	HUS2_VP1_MQ41_ID	AT%MB2524	:REAL;	(*	HUS2_VP1_MQ41_ID	AS01	GVL.HUS2_VP1_MQ41_ID	REAL							Mätar-ID VP1-MQ41			*)
	HUS2_VP1_MQ41_GT41_MV	AT%MB2528	:REAL;	(*	HUS2_VP1_MQ41_GT41_MV	AS01	GVL.HUS2_VP1_MQ41_GT41_MV	REAL	-50	150	-50	150	°C	0.0	Framledningstemperatur fjärrvärme			*)					
	HUS2_VP1_MQ41_GT42_MV	AT%MB2532	:REAL;	(*	HUS2_VP1_MQ41_GT42_MV	AS01	GVL.HUS2_VP1_MQ41_GT42_MV	REAL	-50	150	-50	150	°C	0.0	Returtemperatur fjärrvärme			*)					
	HUS2_VP1_MQ41_DLT	AT%MB2536	:REAL;	(*	HUS2_VP1_MQ41_DLT	AS01	GVL.HUS2_VP1_MQ41_DLT	REAL	-50	150	-50	150	°C	0.0	Temperaturdifferens fjärrvärme			*)					
	HUS2_VP1_MQ41_P	AT%MB2540	:REAL;	(*	HUS2_VP1_MQ41_P	AS01	GVL.HUS2_VP1_MQ41_P	REAL	0	1000	0	1000	Kw	0.0	Momentant effektuttag			*)					
	HUS2_VP1_MQ41_Q	AT%MB2544	:REAL;	(*	HUS2_VP1_MQ41_Q	AS01	GVL.HUS2_VP1_MQ41_Q	REAL	0				m3/h	0.0	Momentant flöde			*)					
	HUS2_VP1_MQ41_E	AT%MB2548	:REAL;	(*	HUS2_VP1_MQ41_E	AS01	GVL.HUS2_VP1_MQ41_E	REAL	0				MWh	0.0	Total energiförbrukning			*)					
																							
	HUS2_VS1_GT11_BB	AT%MB2552	:REAL;	(*	HUS2_VS1_GT11_BB	AS01	GVL.HUS2_VS1_GT11_BB	REAL	0	150	0	150	°C	0.0	Beräknat börvärde framledningstemperatur			*)
	HUS2_VP1_MQ41_BB	AT%MB2556	:REAL;	(*	HUS2_VP1_MQ41_BB	AS01	GVL.HUS2_VP1_MQ41_BB	REAL	0	500	0	500	kWh	0.0	Beräknad maxeffekt			*)				

																							
																							

																						
																						


																					

END_VAR

(* Global variable list: HUS2/VS30/HUS2_VS30_INST *)
VAR_GLOBAL PERSISTENT


					(*	Name	Device	Address	Data type	Rawmin	Rawmax	Engmin	Engmax	Unit	Format	Description	Alarmoptions	Trendoptions	*)
																								
		HUS2_VS30_GT11_UX1	AT%MB2700	:REAL;	(*	HUS2_VS30_GT11_UX1	AS01	GVL.HUS2_VS30_GT11_UX1	REAL	-50	150	-50	150	°C	0.0	Utetemp. kompenserad kurva Brytpunkt X1			*)					
		HUS2_VS30_GT11_UX2	AT%MB2704	:REAL;	(*	HUS2_VS30_GT11_UX2	AS01	GVL.HUS2_VS30_GT11_UX2	REAL	-50	150	-50	150	°C	0.0	Utetemp. kompenserad kurva Brytpunkt X2			*)					
		HUS2_VS30_GT11_UX3	AT%MB2708	:REAL;	(*	HUS2_VS30_GT11_UX3	AS01	GVL.HUS2_VS30_GT11_UX3	REAL	-50	150	-50	150	°C	0.0	Utetemp. kompenserad kurva Brytpunkt X3			*)					
		HUS2_VS30_GT11_UX4	AT%MB2712	:REAL;	(*	HUS2_VS30_GT11_UX4	AS01	GVL.HUS2_VS30_GT11_UX4	REAL	-50	150	-50	150	°C	0.0	Utetemp. kompenserad kurva Brytpunkt X4			*)					
		HUS2_VS30_GT11_UX5	AT%MB2716	:REAL;	(*	HUS2_VS30_GT11_UX5	AS01	GVL.HUS2_VS30_GT11_UX5	REAL	-50	150	-50	150	°C	0.0	Utetemp. kompenserad kurva Brytpunkt X5			*)					
		HUS2_VS30_GT11_UY1	AT%MB2720	:REAL;	(*	HUS2_VS30_GT11_UY1	AS01	GVL.HUS2_VS30_GT11_UY1	REAL	0	150	0	150	°C	0.0	Utetemp. kompenserad kurva Brytpunkt Y1			*)					
		HUS2_VS30_GT11_UY2	AT%MB2724	:REAL;	(*	HUS2_VS30_GT11_UY2	AS01	GVL.HUS2_VS30_GT11_UY2	REAL	0	150	0	150	°C	0.0	Utetemp. kompenserad kurva Brytpunkt Y2			*)					
		HUS2_VS30_GT11_UY3	AT%MB2728	:REAL;	(*	HUS2_VS30_GT11_UY3	AS01	GVL.HUS2_VS30_GT11_UY3	REAL	0	150	0	150	°C	0.0	Utetemp. kompenserad kurva Brytpunkt Y3			*)					
		HUS2_VS30_GT11_UY4	AT%MB2732	:REAL;	(*	HUS2_VS30_GT11_UY4	AS01	GVL.HUS2_VS30_GT11_UY4	REAL	0	150	0	150	°C	0.0	Utetemp. kompenserad kurva Brytpunkt Y4			*)					
		HUS2_VS30_GT11_UY5	AT%MB2736	:REAL;	(*	HUS2_VS30_GT11_UY5	AS01	GVL.HUS2_VS30_GT11_UY5	REAL	0	150	0	150	°C	0.0	Utetemp. kompenserad kurva Brytpunkt Y5			*)					
		HUS2_VS30_GT11_UMIN	AT%MB2740	:REAL;	(*	HUS2_VS30_GT11_UMIN	AS01	GVL.HUS2_VS30_GT11_UMIN	REAL	0	150	0	150	°C	0.0	Utetemp. kompenserad kurva Min-begränsning			*)					
		HUS2_VS30_GT11_UMAX	AT%MB2744	:REAL;	(*	HUS2_VS30_GT11_UMAX	AS01	GVL.HUS2_VS30_GT11_UMAX	REAL	0	150	0	150	°C	0.0	Utetemp. kompenserad kurva Max-begränsning			*)					
																								
		HUS2_VS30_GT11_CP	AT%MB2748	:REAL;	(*	HUS2_VS30_GT11_CPV	AS01	GVL.HUS2_VS30_GT11_CP	REAL	0	10	0	10		0.0	P-parameter			*)					
		HUS2_VS30_GT11_CI	AT%MB2752	:REAL;	(*	HUS2_VS30_GT11_CIV	AS01	GVL.HUS2_VS30_GT11_CI	REAL	0	900	0	900	Sek		I-Tid 			*)
		HUS2_VS30_GT11_CD	AT%MB2756	:REAL;	(*	HUS2_VS30_GT11_CDV	AS01	GVL.HUS2_VS30_GT11_CD	REAL	0	900	0	900	Sek		D-tid 			*)
		HUS2_VS30_GT11_CS	AT%MB2760	:REAL;	(*	HUS2_VS30_GT11_CSV	AS01	GVL.HUS2_VS30_GT11_CS	REAL	0	900	0	900	Sek		Samplingstid			*)
		HUS2_VS30_GT11_CZ	AT%MB2764	:REAL;	(*	HUS2_VS30_GT11_CZV	AS01	GVL.HUS2_VS30_GT11_CZ	REAL	-10	10	-10	10	°C	0.0	Dödband regulator			*)					
																								
		HUS2_VS30_SO1_MAN	AT%MB2768	:INT;	(*	HUS2_VS30_SO1_MAN	AS01	GVL.HUS2_VS30_SO1_MAN	INT	0	2	0	2			Manuell styrning system VS30. 0=Auto, 1=Manuell från, 2=Manuell till			*)					
		HUS2_VS30_PV01_MAN	AT%MB2770	:INT;	(*	HUS2_VS30_PV01_MAN	AS01	GVL.HUS2_VS30_PV01_MAN	INT	0	2	0	2			Manuell styrning crikulationspump 0=Auto,1=Från,2=Till			*)					
		HUS2_VS30_SV21_MAN1	AT%MB2772	:INT;	(*	HUS2_VS30_SV21_MAN	AS01	GVL.HUS2_VS30_SV21_MAN	INT	0	1	0	1			Manuell styrning ventilställdon 0=Auto,1=Hand			*)					
		HUS2_VS30_SV21_RMAN	AT%MB2776	:REAL;	(*	HUS2_VS30_SV21_RMAN	AS01	GVL.HUS2_VS30_SV21_RMAN	REAL	0	100	0	100	%		Manuell styrsignal ventilställdon			*)					
																								
		HUS2_VS30_SO1_FLM	AT%MB2780	:INT;	(*	HUS2_VS30_SO1_FLM	AS01	GVL.HUS2_VS30_SO1_FLM	INT	0	3600	0	3600	Min		Larmfördröjning serviceomkopplare ej i läge AUTO			*)					
		HUS2_VS30_PV01_FLM	AT%MB2782	:INT;	(*	HUS2_VS30_PV01_FLM	AS01	GVL.HUS2_VS30_PV01_FLM	INT	0	3600	0	3600	Min		Larmfördröjning cirkulationspump ej i AUTO			*)					
		HUS2_VS30_SV21_FLM	AT%MB2784	:INT;	(*	HUS2_VS30_SV21_FLM	AS01	GVL.HUS2_VS30_SV21_FLM	INT	0	3600	0	3600	Min		Larmfördröjning ventilställdon ej i AUTO			*)					
		HUS2_VS30_PV01_FLD	AT%MB2786	:INT;	(*	HUS2_VS30_PV01_FLD	AS01	GVL.HUS2_VS30_PV01_FLD	INT	0	120	0	120	Sek		Larmfördröjning driftfel cirkulationspump			*)					
																								
		HUS2_VS30_GT11_GAVH	AT%MB2788	:REAL;	(*	HUS2_VS30_GT11_GAVH	AS01	GVL.HUS2_VS30_GT11_GAVH	REAL	-20	20	-20	20	°C	0.0	Gränsavvikelse hög framledningstemperatur			*)					
		HUS2_VS30_GT11_GAVL	AT%MB2792	:REAL;	(*	HUS2_VS30_GT11_GAVL	AS01	GVL.HUS2_VS30_GT11_GAVL	REAL	-20	20	-20	20	°C	0.0	Gränsavvikelse låg framledningstemperatur			*)					
		HUS2_VS30_GT11_FLAH	AT%MB2796	:INT;	(*	HUS2_VS30_GT11_FLAH	AS01	GVL.HUS2_VS30_GT11_FLAH	INT	0	3600	0	3600	Min		Larmfördröjning hög framledningstemperatur			*)					
		HUS2_VS30_GT11_FLAL	AT%MB2798	:INT;	(*	HUS2_VS30_GT11_FLAL	AS01	GVL.HUS2_VS30_GT11_FLAL	INT	0	3600	0	3600	Min		Lamfördröjning låg framledningstemperatur			*)					


																								

																								
		HUS2_VS30_GT11_KRV	AT%MB2816	:REAL;	(*	HUS2_VS30_GT11_KRV	AS01	GVL.HUS2_VS30_GT11_KRV	REAL	-10	10	-10	10	°C	0.0	Kalibreringsvärde framledningsgivare			*)					
		HUS2_VS30_GT41_KRV	AT%MB2820	:REAL;	(*	HUS2_VS30_GT41_KRV	AS01	GVL.HUS2_VS30_GT41_KRV	REAL	-10	10	-10	10	°C	0.0	Kalibreringsvärde returgivare			*)					
																								
		HUS2_VS30_GT11_X1	AT%MB2824	:REAL;	(*	HUS2_VS30_GT11_X1	AS01	GVL.HUS2_VS30_GT11_X1	REAL	-50	150	-50	150	°C	0.0	Effektbegränsning kurva Brytpunkt X1			*)
		HUS2_VS30_GT11_X2	AT%MB2828	:REAL;	(*	HUS2_VS30_GT11_X2	AS01	GVL.HUS2_VS30_GT11_X2	REAL	-50	150	-50	150	°C	0.0	Effektbegränsning kurva Brytpunkt X2			*)	
		HUS2_VS30_GT11_X3	AT%MB2832	:REAL;	(*	HUS2_VS30_GT11_X3	AS01	GVL.HUS2_VS30_GT11_X3	REAL	-50	150	-50	150	°C	0.0	Effektbegränsning kurva Brytpunkt X3			*)	
		HUS2_VS30_GT11_X4	AT%MB2836	:REAL;	(*	HUS2_VS30_GT11_X4	AS01	GVL.HUS2_VS30_GT11_X4	REAL	-50	150	-50	150	°C	0.0	Effektbegränsning kurva Brytpunkt X4			*)	
		HUS2_VS30_GT11_X5	AT%MB2840	:REAL;	(*	HUS2_VS30_GT11_X5	AS01	GVL.HUS2_VS30_GT11_X5	REAL	-50	150	-50	150	°C	0.0	Effektbegränsning kurva Brytpunkt X5			*)	
		HUS2_VS30_GT11_Y1	AT%MB2844	:REAL;	(*	HUS2_VS30_GT11_Y1	AS01	GVL.HUS2_VS30_GT11_Y1	REAL	0	150	0	150	°C	0.0	Effektbegränsning kurva Brytpunkt Y1			*)	
		HUS2_VS30_GT11_Y2	AT%MB2848	:REAL;	(*	HUS2_VS30_GT11_Y2	AS01	GVL.HUS2_VS30_GT11_Y2	REAL	0	150	0	150	°C	0.0	Effektbegränsning kurva Brytpunkt Y2			*)	
		HUS2_VS30_GT11_Y3	AT%MB2852	:REAL;	(*	HUS2_VS30_GT11_Y3	AS01	GVL.HUS2_VS30_GT11_Y3	REAL	0	150	0	150	°C	0.0	Effektbegränsning kurva Brytpunkt Y3			*)	
		HUS2_VS30_GT11_Y4	AT%MB2856	:REAL;	(*	HUS2_VS30_GT11_Y4	AS01	GVL.HUS2_VS30_GT11_Y4	REAL	0	150	0	150	°C	0.0	Effektbegränsning kurva Brytpunkt Y4			*)	
		HUS2_VS30_GT11_Y5	AT%MB2860	:REAL;	(*	HUS2_VS30_GT11_Y5	AS01	GVL.HUS2_VS30_GT11_Y5	REAL	0	150	0	150	°C	0.0	Effektbegränsning kurva Brytpunkt Y5			*)	
		HUS2_VS30_GT11_MIN	AT%MB2864	:REAL;	(*	HUS2_VS30_GT11_MIN	AS01	GVL.HUS2_VS30_GT11_MIN	REAL	0	150	0	150	°C	0.0	Effektbegränsning kurva Min-begränsning			*)
		HUS2_VS30_GT11_MAX	AT%MB2868	:REAL;	(*	HUS2_VS30_GT11_MAX	AS01	GVL.HUS2_VS30_GT11_MAX	REAL	0	150	0	150	°C	0.0	Effektbegränsning kurva Max-begränsning			*)	

																				

																								
																								
																								
																								
																								
																								
																								


END_VAR
																
																

(* Global variable list: HUS2/VS30/HUS2_VS30_LARM *)
VAR_GLOBAL



																						
	HUS2_VS30_SO1_LM	AT%MX2910.0	:BOOL; 	(*	HUS2_VS30_SO1_LM	AS01	GVL.HUS2_VS30_SO1_LM	DIGITAL	0	0	0	0			Serviceomkopplare ej i läge AUTO	p:C		*)				
	HUS2_VS30_PV01_LM	AT%MX2910.1	:BOOL; 	(*	HUS2_VS30_PV01_LM	AS01	GVL.HUS2_VS30_PV01_LM	DIGITAL	0	0	0	0			Cirkulationspump ej i AUTO	p:B		*)				
	HUS2_VS30_SV21_LM	AT%MX2910.2	:BOOL; 	(*	HUS2_VS30_SV21_LM	AS01	GVL.HUS2_VS30_SV21_LM	DIGITAL	0	0	0	0			Ventilställdon ej i AUTO	p:B		*)				
	HUS2_VS30_PV01_LD	AT%MX2910.3	:BOOL; 	(*	HUS2_VS30_PV01_LD	AS01	GVL.HUS2_VS30_PV01_LD	DIGITAL	0	0	0	0			Driftfel cirkulationspump	p:B		*)				
	HUS2_VS30_GT11_LG	AT%MX2910.4	:BOOL; 	(*	HUS2_VS30_GT11_LG	AS01	GVL.HUS2_VS30_GT11_LG	DIGITAL	0	0	0	0			Givarfel framledningsgivare	p:B		*)				
	HUS2_VS30_GT41_LG	AT%MX2910.5	:BOOL; 	(*	HUS2_VS30_GT41_LG	AS01	GVL.HUS2_VS30_GT41_LG	DIGITAL	0	0	0	0			Givarfel returgivare	p:B		*)
	HUS2_VS30_GT11_LAH	AT%MX2910.6	:BOOL; 	(*	HUS2_VS30_GT11_LAH	AS01	GVL.HUS2_VS30_GT11_LAH	DIGITAL	0	0	0	0			Larmavvikelse hög framledningstemp	p:B		*)				
	HUS2_VS30_GT11_LAL	AT%MX2910.7	:BOOL; 	(*	HUS2_VS30_GT11_LAL	AS01	GVL.HUS2_VS30_GT11_LAL	DIGITAL	0	0	0	0			Larmavvikelse låg framledningstemp	p:B		*)				



																						
	HUS2_VS30_PV01_ACK	AT%MX2918.0	:BOOL; 	(*	HUS2_VS30_PV01_ACK	AS01	GVL.HUS2_VS30_PV01_ACK	DIGITAL	0	0	0	0			Larmkvittens pump			*)				
																						
																						
																						
																						

																						



END_VAR

(* Global variable list: HUS2/VS30/HUS2_VS30_OVRIGT *)
VAR_GLOBAL



																						
	HUS2_VS30_SO1_IH	AT%MX2920.0	:BOOL;	(*	HUS2_VS30_SO1_IH	AS01	GVL.HUS2_VS30_SO1_IH	DIGITAL	0	0	0	0			Serviceomkopplare ej i AUTO			*)				
	HUS2_VS30_SO1_IA	AT%MX2920.1	:BOOL;	(*	HUS2_VS30_SO1_IA	AS01	GVL.HUS2_VS30_SO1_IA	DIGITAL	0	0	0	0			Serviceomkopplare i läge AUTO			*)				
	HUS2_VS30_SO1_IF	AT%MX2920.2	:BOOL;	(*	HUS2_VS30_SO1_IF	AS01	GVL.HUS2_VS30_SO1_IF	DIGITAL	0	0	0	0			Serviceomkopplare i läge 0			*)				
	HUS2_VS30_SO1_IT	AT%MX2920.3	:BOOL;	(*	HUS2_VS30_SO1_IT	AS01	GVL.HUS2_VS30_SO1_IT	DIGITAL	0	0	0	0			Serviceomkopplare i läge HAND TILL			*)				


																						
																						
																						
																						
																						

																						
																						
																						
																						
	HUS2_VS30_GT11_BB	AT%MB2952	:REAL;	(*	HUS2_VS30_GT11_BB	AS01	GVL.HUS2_VS30_GT11_BB	REAL	0	150	0	150	°C	0.0	Beräknat börvärde framledningstemperatur			*)				
	HUS2_VS30_GT11_BB1	AT%MB2956	:REAL;	(*	HUS2_VS30_GT11_BB1	AS01	GVL.HUS2_VS30_GT11_BB1	REAL	0	150	0	150	°C	0.0	Beräknad förskjutning framledningstemperatur			*)

																						
																						

																						

																						

																					

END_VAR

(* Global variable list: HUS2/VV1/HUS2_VV1_INST *)
VAR_GLOBAL PERSISTENT
				(*	Name	Device	Address	Data type	Rawmin	Rawmax	Engmin	Engmax	Unit	Format	Description	Alarmoptions	Trendoptions	*)
																		

																		
	HUS2_VV1_SO1_MAN	AT%MB3264	:INT;	(*	HUS2_VV1_SO1_MAN	AS01	GVL.HUS2_VV1_SO1_MAN	INT	0	2	0	2			Manuell styrning system VV1. 0=Auto, 1=Manuell från, 2=Manuell till			*)
	HUS2_VVC1_PC01_MAN	AT%MB3266	:INT;	(*	HUS2_VVC1_PC01_MAN	AS01	GVL.HUS2_VVC1_PC01_MAN	INT	0	2	0	2			Manuell styrning crikulationspump 0=Auto,1=Från,2=Till			*)
	HUS2_VV1_SV11_MAN1	AT%MB3268	:INT;	(*	HUS2_VV1_SV11_MAN	AS01	GVL.HUS2_VV1_SV11_MAN	INT	0	1	0	1			Manuell styrning ventilställdon 0=Auto,1=Hand			*)
	HUS2_VV1_SV11_RMAN	AT%MB3272	:REAL;	(*	HUS2_VV1_SV11_RMAN	AS01	GVL.HUS2_VV1_SV11_RMAN	REAL	0	100	0	100	%		Manuell styrsignal ventilställdon			*)
	HUS2_VV1_SO1_FLM	AT%MB3276	:INT;	(*	HUS2_VV1_SO1_FLM	AS01	GVL.HUS2_VV1_SO1_FLM	INT	0	3600	0	3600	Min		Larmfördröjning serviceomkopplare ej i läge AUTO			*)
	HUS2_VVC1_PC01_FLM	AT%MB3278	:INT;	(*	HUS2_VVC1_PC01_FLM	AS01	GVL.HUS2_VVC1_PC01_FLM	INT	0	3600	0	3600	Min		Larmfördröjning cirkulationspump ej i AUTO			*)
	HUS2_VV1_SV11_FLM	AT%MB3280	:INT;	(*	HUS2_VV1_SV11_FLM	AS01	GVL.HUS2_VV1_SV11_FLM	INT	0	3600	0	3600	Min		Larmfördröjning ventilställdon ej i AUTO			*)
	HUS2_VVC1_PC01_FLD	AT%MB3282	:INT;	(*	HUS2_VVC1_PC01_FLD	AS01	GVL.HUS2_VVC1_PC01_FLD	INT	0	120	0	120	Sek		Larmfördröjning driftfel cirkulationspump			*)


	HUS2_VV1_GT11_CP	AT%MB3284	:REAL;	(*	HUS2_VV1_GT11_CPV	AS01	GVL.HUS2_VV1_GT11_CP	REAL	0	10	0	10		0.0	P-parameter			*)
	HUS2_VV1_GT11_CI	AT%MB3288	:REAL;	(*	HUS2_VV1_GT11_CIV	AS01	GVL.HUS2_VV1_GT11_CI	REAL	0	900	0	900	Sek		I-Tid 			*)
	HUS2_VV1_GT11_CD	AT%MB3292	:REAL;	(*	HUS2_VV1_GT11_CDV	AS01	GVL.HUS2_VV1_GT11_CD	REAL	0	900	0	900	Sek		D-tid 			*)
	HUS2_VV1_GT11_CS	AT%MB3296	:REAL;	(*	HUS2_VV1_GT11_CSV	AS01	GVL.HUS2_VV1_GT11_CS	REAL	0	900	0	900	Sek		Samplingstid			*)
	HUS2_VV1_GT11_CZ	AT%MB3300	:REAL;	(*	HUS2_VV1_GT11_CZV	AS01	GVL.HUS2_VV1_GT11_CZ	REAL	-10	10	-10	10	°C	0.0	Dödband regulator			*)
																		
																		
	HUS2_VV1_GT11_GAVH	AT%MB3304	:REAL;	(*	HUS2_VV1_GT11_GAVH	AS01	GVL.HUS2_VV1_GT11_GAVH	REAL	-20	20	-20	20	°C	0.0	Gränsavvikelse hög framledningstemperatur			*)
	HUS2_VV1_GT11_GAVL	AT%MB3308	:REAL;	(*	HUS2_VV1_GT11_GAVL	AS01	GVL.HUS2_VV1_GT11_GAVL	REAL	-20	20	-20	20	°C	0.0	Gränsavvikelse låg framledningstemperatur			*)
	HUS2_VV1_GT11_FLAH	AT%MB3312	:INT;	(*	HUS2_VV1_GT11_FLAH	AS01	GVL.HUS2_VV1_GT11_FLAH	INT	0	3600	0	3600	Min		Larmfördröjning hög framledningstemperatur			*)
	HUS2_VV1_GT11_FLAL	AT%MB3316	:INT;	(*	HUS2_VV1_GT11_FLAL	AS01	GVL.HUS2_VV1_GT11_FLAL	INT	0	3600	0	3600	Min		Lamfördröjning låg framledningstemperatur			*)
	HUS2_VVC1_GT41_GVL	AT%MB3320	:REAL;	(*	HUS2_VVC1_GT41_GVL	AS01	GVL.HUS2_VVC1_GT41_GVL	REAL	0	150	0	150	°C	0.0	Gränsvärde låg VVC-temperatur			*)
	HUS2_VVC1_GT41_FLG	AT%MB3324	:INT;	(*	HUS2_VVC1_GT41_FLG	AS01	GVL.HUS2_VVC1_GT41_FLG	INT	0	3600	0	3600	Min		Lamfördröjning låg VVC-temperatur			*)
																		
																		

	HUS2_VV1_GT11_KRV	AT%MB3332	:REAL;	(*	HUS2_VV1_GT11_KRV	AS01	GVL.HUS2_VV1_GT11_KRV	REAL	-10	10	-10	10	°C	0.0	Kalibreringsvärde framledningsgivare			*)
	HUS2_VVC1_GT41_KRV	AT%MB3336	:REAL;	(*	HUS2_VVC1_GT41_KRV	AS01	GVL.HUS2_VVC1_GT41_KRV	REAL	-10	10	-10	10	°C	0.0	Kalibreringsvärde returgivare VVC			*)
	HUS2_KV1_GT41_KRV	AT%MB3340	:REAL;	(*	HUS2_KV1_GT41_KRV	AS01	GVL.HUS2_KV1_GT41_KRV	REAL	-10	10	-10	10	°C	0.0	Kalibreringsvärde kallvattengivare			*)

																		



	END_VAR
																
																

(* Global variable list: HUS2/VV1/HUS2_VV1_LARM *)
VAR_GLOBAL


																					
	HUS2_VV1_SO1_LM	AT%MX3360.0	:BOOL; 	(*	HUS2_VV1_SO1_LM	AS01	GVL.HUS2_VV1_SO1_LM	DIGITAL	0	0	0	0			Serviceomkopplare ej i läge TILL	p:C		*)			
	HUS2_VVC1_PC01_LM	AT%MX3360.1	:BOOL; 	(*	HUS2_VVC1_PC01_LM	AS01	GVL.HUS2_VVC1_PC01_LM	DIGITAL	0	0	0	0			Cirkulationspump ej i AUTO	p:B		*)			
	HUS2_VV1_SV11_LM	AT%MX3360.2	:BOOL; 	(*	HUS2_VV1_SV11_LM	AS01	GVL.HUS2_VV1_SV11_LM	DIGITAL	0	0	0	0			Ventilställdon ej i AUTO	p:B		*)			
	HUS2_VVC1_PC01_LD	AT%MX3360.3	:BOOL; 	(*	HUS2_VVC1_PC01_LD	AS01	GVL.HUS2_VVC1_PC01_LD	DIGITAL	0	0	0	0			Driftfel cirkulationspump	p:B		*)			
	HUS2_VV1_GT11_LG	AT%MX3360.4	:BOOL; 	(*	HUS2_VV1_GT11_LG	AS01	GVL.HUS2_VV1_GT11_LG	DIGITAL	0	0	0	0			Givarfel framledningsgivare	p:B		*)			
	HUS2_VVC1_GT41_LG	AT%MX3360.5	:BOOL; 	(*	HUS2_VVC1_GT41_LG	AS01	GVL.HUS2_VVC1_GT41_LG	DIGITAL	0	0	0	0			Givarfel VVC-givare	p:B		*)			
	HUS2_KV1_GT41_LG	AT%MX3360.6	:BOOL; 	(*	HUS2_KV1_GT41_LG	AS01	GVL.HUS2_KV1_GT41_LG	DIGITAL	0	0	0	0			Givarfel kallvattengivare	p:B		*)			
	HUS2_VV1_GT11_LAH	AT%MX3360.7	:BOOL; 	(*	HUS2_VV1_GT11_LAH	AS01	GVL.HUS2_VV1_GT11_LAH	DIGITAL	0	0	0	0			Larmavvikelse hög framledningstemp	p:B		*)			
	HUS2_VV1_GT11_LAL	AT%MX3361.0	:BOOL; 	(*	HUS2_VV1_GT11_LAL	AS01	GVL.HUS2_VV1_GT11_LAL	DIGITAL	0	0	0	0			Larmavvikelse låg framledningstemp	p:B		*)			
	HUS2_VVC1_GT41_LL	AT%MX3361.1	:BOOL; 	(*	HUS2_VVC1_GT41_LL	AS01	GVL.HUS2_VVC1_GT41_LL	DIGITAL	0	0	0	0			Låg VVC-temperatur	p:B		*)			
	HUS2_VV1_MQ41_L	AT%MX3361.2	:BOOL; 	(*	HUS2_VV1_MQ41_L	AS01	GVL.HUS2_VV1_MQ41_L	DIGITAL	0	0	0	0			Summalarm energimätare	p:B		*)			
	HUS2_VV1_MQ41_LC	AT%MX3361.3	:BOOL; 	(*	HUS2_VV1_MQ41_LC	AS01	GVL.HUS2_VV1_MQ41_LC	DIGITAL	0	0	0	0			Kommunikationsfel energimätare	p:B		*)			
	HUS2_VVC1_MQ41_L	AT%MX3361.4	:BOOL; 	(*	HUS2_VP1_MQ41_L	AS01	GVL.HUS2_VP1_MQ41_L	DIGITAL	0	0	0	0			Summalarm energimätare	p:B		*)			
	HUS2_VVC1_MQ41_LC	AT%MX3361.5	:BOOL; 	(*	HUS2_VP1_MQ41_LC	AS01	GVL.HUS2_VP1_MQ41_LC	DIGITAL	0	0	0	0			Kommunikationsfel energimätare	p:B		*)			
	HUS2_KV1_MF41_L	AT%MX3361.6	:BOOL; 	(*	HUS2_KV1_MF41_L	AS01	GVL.HUS2_KV1_MF41_L	DIGITAL	0	0	0	0			Summalarm kallvattenmätare	p:B		*)
	HUS2_KV1_MF41_LC	AT%MX3361.7	:BOOL; 	(*	HUS2_KV1_MF41_LC	AS01	GVL.HUS2_KV1_MF41_LC	DIGITAL	0	0	0	0			Kommunikationsfel kallvattenmätare	p:B		*)
	HUS2_KV1_MF42_LC	AT%MX3362.0	:BOOL; 	(*	HUS2_KV1_MF42_LC	AS01	HUS2_VV1_LARM.HUS2_KV1_MF42_LC	DIGITAL	0	0	0	0			Kommunikationsfel kallvattenmätare	p:B		*)
																					

																					
																					
	HUS2_VVC1_PC01_ACK	AT%MX3363.0	:BOOL; 	(*	HUS2_VVC1_PC01_ACK	AS01	GVL.HUS2_VVC1_PC01_ACK	DIGITAL	0	0	0	0			Larmkvittens pump			*)			
																					
																					




END_VAR

(* Global variable list: HUS2/VV1/HUS2_VV1_OVRIGT *)
VAR_GLOBAL

																				
	HUS2_VV1_SO1_IF	AT%MX3370.0	:BOOL;	(*	HUS2_VV1_SO1_IF	AS01	GVL.HUS2_VV1_SO1_IF	DIGITAL	0	0	0	0			Serviceomkopplare i läge 0			*)		
	HUS2_VV1_SO1_IT	AT%MX3370.1	:BOOL;	(*	HUS2_VV1_SO1_IT	AS01	GVL.HUS2_VV1_SO1_IT	DIGITAL	0	0	0	0			Serviceomkopplare i läge TILL			*)		

																				
																				
																				
																				
	HUS2_VV1_MQ41_ID	AT%MB3376	:REAL;	(*	HUS2_VV1_MQ41_ID	AS01	GVL.HUS2_VV1_MQ41_ID	REAL							Mätar-ID VV1-MQ41			*)
	HUS2_VV1_MQ41_GT41_MV	AT%MB3380	:REAL;	(*	HUS2_VV1_MQ41_GT41_MV	AS01	GVL.HUS2_VV1_MQ41_GT41_MV	REAL	-50	150	-50	150	°C	0.0	Framledningstemperatur			*)		
	HUS2_VV1_MQ41_GT42_MV	AT%MB3384	:REAL;	(*	HUS2_VV1_MQ41_GT42_MV	AS01	GVL.HUS2_VV1_MQ41_GT42_MV	REAL	-50	150	-50	150	°C	0.0	Returtemperatur			*)		
	HUS2_VV1_MQ41_DLT	AT%MB3388	:REAL;	(*	HUS2_VV1_MQ41_DLT	AS01	GVL.HUS2_VV1_MQ41_DLT	REAL	-50	150	-50	150	°C	0.0	Temperaturdifferens			*)		
	HUS2_VV1_MQ41_P	AT%MB3392	:REAL;	(*	HUS2_VV1_MQ41_P	AS01	GVL.HUS2_VV1_MQ41_P	REAL	0	1000	0	1000	Kw	0.0	Momentant effektuttag			*)
	HUS2_VV1_MQ41_Q	AT%MB3396	:REAL;	(*	HUS2_VV1_MQ41_Q	AS01	GVL.HUS2_VV1_MQ41_Q	REAL	0				m3/h	0.0	Momentant flöde			*)
	HUS2_VV1_MQ41_E	AT%MB3400	:REAL;	(*	HUS2_VV1_MQ41_E	AS01	GVL.HUS2_VV1_MQ41_E	REAL	0				MWh	0.0	Total energiförbrukning			*)
	HUS2_VVC1_MQ41_ID	AT%MB3404	:REAL;	(*	HUS2_VVC1_MQ41_ID	AS01	GVL.HUS2_VVC1_MQ41_ID	REAL							Mätar-ID VVC1-MQ41			*)
	HUS2_VVC1_MQ41_GT41_MV	AT%MB3408	:REAL;	(*	HUS2_VVC1_MQ41_GT41_MV	AS01	GVL.HUS2_VVC1_MQ41_GT41_MV	REAL	-50	150	-50	150	°C	0.0	Framledningstemperatur			*)		
	HUS2_VVC1_MQ41_GT42_MV	AT%MB3412	:REAL;	(*	HUS2_VVC1_MQ41_GT42_MV	AS01	GVL.HUS2_VVC1_MQ41_GT42_MV	REAL	-50	150	-50	150	°C	0.0	Returtemperatur			*)		
	HUS2_VVC1_MQ41_DLT	AT%MB3416	:REAL;	(*	HUS2_VVC1_MQ41_DLT	AS01	GVL.HUS2_VVC1_MQ41_DLT	REAL	-50	150	-50	150	°C	0.0	Temperaturdifferens			*)
	HUS2_VVC1_MQ41_P	AT%MB3420	:REAL;	(*	HUS2_VVC1_MQ41_P	AS01	GVL.HUS2_VVC1_MQ41_P	REAL	0	1000	0	1000	Kw	0.0	Momentant effektuttag			*)
	HUS2_VVC1_MQ41_Q	AT%MB3424	:REAL;	(*	HUS2_VVC1_MQ41_Q	AS01	GVL.HUS2_VVC1_MQ41_Q	REAL	0				m3/h	0.0	Momentant flöde			*)
	HUS2_VVC1_MQ41_E	AT%MB3428	:REAL;	(*	HUS2_VVC1_MQ41_E	AS01	GVL.HUS2_VVC1_MQ41_E	REAL	0				MWh	0.0	Total energiförbrukning			*)
	HUS2_KV1_MF41_ID	AT%MB3432	:REAL;	(*	HUS2_KV1_MF41_ID	AS01	GVL.HUS2_KV1_MF41_ID	REAL							Mätar-ID KV1-MF41			*)
	HUS2_KV1_MF41_Q	AT%MB3436	:REAL;	(*	HUS2_KV1_MF41_Q		HUS2_KV1_MF41_Q	REAL	0	10000000	0	10000000	m3		Volym			*)
	HUS2_KV1_MF42_Q	AT%MB3440	:REAL;	(*	HUS2_KV1_MF42_Q	AS01	HUS2_VV1_OVRIGTHUS2_KV1_MF42_Q	REAL	0	10000000	0	10000000	m3		Volym			*)
																				
																				
																				





																					

END_VAR

(* Global variable list: HUS3/AL02/HUS3_AL02_IO_Hardvara *)
VAR_GLOBAL

										
	(* Digitala in, KL1488  *)									
	(*Kort1*)									
		AL02_Kort01_DI01				AT %I*			:BOOL;	
		AL02_Kort01_DI02				AT %I*			:BOOL;	
		AL02_Kort01_DI03				AT %I*			:BOOL;	
		AL02_Kort01_DI04				AT %I*			:BOOL;	
		AL02_Kort01_DI05				AT %I*			:BOOL;	
		AL02_Kort01_DI06				AT %I*			:BOOL;	
		AL02_Kort01_DI07				AT %I*			:BOOL;	
		AL02_Kort01_DI08				AT %I*			:BOOL;	
										
										
	(* Digitala in, KL1488  *)									
	(*Kort2*)									
		AL02_Kort02_DI01				AT %I*			:BOOL;	
		AL02_Kort02_DI02				AT %I*			:BOOL;	
		AL02_Kort02_DI03				AT %I*			:BOOL;	
		AL02_Kort02_DI04				AT %I*			:BOOL;	
		AL02_Kort02_DI05				AT %I*			:BOOL;	
		AL02_Kort02_DI06				AT %I*			:BOOL;	
		AL02_Kort02_DI07				AT %I*			:BOOL;	
		AL02_Kort02_DI08				AT %I*			:BOOL;	
										
										
	(* Digital Ut, KL2408 *)									
	(*Kort3*)									
		AL02_Kort03_DU01				AT %Q*			:BOOL;
		AL02_Kort03_DU02				AT %Q*			:BOOL;	
		AL02_Kort03_DU03				AT %Q*			:BOOL;	
		AL02_Kort03_DU04				AT %Q*			:BOOL;	
		AL02_Kort03_DU05				AT %Q*			:BOOL;	
		AL02_Kort03_DU06				AT %Q*			:BOOL;	
		AL02_Kort03_DU07				AT %Q*			:BOOL;	
		AL02_Kort03_DU08				AT %Q*			:BOOL;	
										
										
										


												

END_VAR

(* Global variable list: HUS3/AL02/HUS3_AL02_IO_Program *)
VAR_GLOBAL


					(*	Name	Device	Address	Data type	Rawmin	Rawmax	Engmin	Engmax	Unit	Format	Description	Alarmoptions	Trendoptions	*)		
	(* Digitala in, KL1488  *)																				
	(*Kort 1*)																				
		HUS3_AL02_FS01_L	AT%MX223.0	:BOOL;	(*	HUS3_AL02_FS01_L	AS01	GVL.HUS3_AL02_FS01_L	DIGITAL	0	0	0	0			Utlöst dvärgbrytare 	p:B		*)		
		HUS3_LB04_HD74_L	AT%MX223.1	:BOOL;	(*	HUS3_LB04_HD74_L	AS01	GVL.HUS3_LB04_HD74_L	DIGITAL	0	0	0	0			Utlöst rökdetektor 	p:A		*)		
		HUS3_LB04_HD74_L1	AT%MX223.2	:BOOL;	(*	HUS3_LB04_HD74_L1	AS01	GVL.HUS3_LB04_HD74_L1	DIGITAL	0	0	0	0			Servicelarm	p:B		*)		
		HUS3_LB04_HD74_L2	AT%MX223.3	:BOOL;	(*	HUS3_LB04_HD74_L2	AS01	GVL.HUS3_LB04_HD74_L2	DIGITAL	0	0	0	0			Fellarm 	p:B		*)		
		HUS3_LB04_BS205_IO	AT%MX223.4	:BOOL;	(*	HUS3_LB04_BS205_IO	AS01	GVL.HUS3_LB04_BS205_IO	DIGITAL	0	0	0	0			Indikering öppet 			*)		
		HUS3_LB04_BS205_IS	AT%MX223.5	:BOOL;	(*	HUS3_LB04_BS205_IS	AS01	GVL.HUS3_LB04_BS205_IS	DIGITAL	0	0	0	0			Indikering stängt 			*)		
		HUS3_LB04_BS206_IO	AT%MX223.6	:BOOL;	(*	HUS3_LB04_BS206_IO	AS01	GVL.HUS3_LB04_BS206_IO	DIGITAL	0	0	0	0			Indikering öppet 			*)		
		HUS3_LB04_BS206_IS	AT%MX223.7	:BOOL;	(*	HUS3_LB04_BS206_IS	AS01	GVL.HUS3_LB04_BS206_IS	DIGITAL	0	0	0	0			Indikering stängt 			*)		
																					
																					
	(* Digitala in, KL1488  *)																				
	(*Kort 2*)																				
		HUS3_LB04_BS207_IO	AT%MX224.0	:BOOL;	(*	HUS3_LB04_BS207_IO	AS01	GVL.HUS3_LB04_BS207_IO	DIGITAL	0	0	0	0			Indikering öppet 	p:A		*)		
		HUS3_LB04_BS207_IS	AT%MX224.1	:BOOL;	(*	HUS3_LB04_BS207_IS	AS01	GVL.HUS3_LB04_BS207_IS	DIGITAL	0	0	0	0			Indikering stängt 	p:B		*)		
		HUS3_AL02_RESERV_DI_KORT02_CH03	AT%MX224.2	:BOOL;	(*											Reserv 			*)		
		HUS3_AL02_RESERV_DI_KORT02_CH04	AT%MX224.3	:BOOL;	(*											Reserv 			*)		
		HUS3_AL02_RESERV_DI_KORT02_CH05	AT%MX224.4	:BOOL;	(*											Reserv 			*)		
		HUS3_AL02_RESERV_DI_KORT02_CH06	AT%MX224.5	:BOOL;	(*											Reserv 			*)		
		HUS3_AL02_RESERV_DI_KORT02_CH07	AT%MX224.6	:BOOL;	(*											Reserv 			*)		
		HUS3_AL02_RESERV_DI_KORT02_CH08	AT%MX224.7	:BOOL;	(*											Reserv 			*)		
																					
																					
	(* Digital Ut, KL2408 *)																				
	(*Kort 3*)																				
		HUS3_LB04_BS205_M	AT%MX225.0	:BOOL;	(*											Manöver			*)		
		HUS3_LB04_BS206_M	AT%MX225.1	:BOOL;	(*											Manöver			*)		
		HUS3_LB04_BS207_M	AT%MX225.2	:BOOL;	(*											Manöver 			*)		
		HUS3_AL02_RESERV_DU_KORT03_CH04	AT%MX225.3	:BOOL;	(*											Reserv 			*)		
		HUS3_AL02_RESERV_DU_KORT03_CH05	AT%MX225.4	:BOOL;	(*											Reserv 			*)		
		HUS3_AL02_RESERV_DU_KORT03_CH06	AT%MX225.5	:BOOL;	(*											Reserv 			*)		
		HUS3_AL02_RESERV_DU_KORT03_CH07	AT%MX225.6	:BOOL;	(*											Reserv 			*)		
		HUS3_AL02_RESERV_DU_KORT03_CH08	AT%MX225.7	:BOOL;	(*											Reserv 			*)		
																					
																					
																					




END_VAR

(* Global variable list: HUS3/AL03/HUS3_AL03_IO_Hardvara *)
VAR_GLOBAL

										
	(* Digitala in, KL1488  *)									
	(*Kort1*)									
		AL03_Kort01_DI01				AT %I*			:BOOL;	
		AL03_Kort01_DI02				AT %I*			:BOOL;	
		AL03_Kort01_DI03				AT %I*			:BOOL;	
		AL03_Kort01_DI04				AT %I*			:BOOL;	
		AL03_Kort01_DI05				AT %I*			:BOOL;	
		AL03_Kort01_DI06				AT %I*			:BOOL;	
		AL03_Kort01_DI07				AT %I*			:BOOL;	
		AL03_Kort01_DI08				AT %I*			:BOOL;	
										
										
	(* Digitala in, KL1488  *)									
	(*Kort2*)									
		AL03_Kort02_DI01				AT %I*			:BOOL;	
		AL03_Kort02_DI02				AT %I*			:BOOL;	
		AL03_Kort02_DI03				AT %I*			:BOOL;	
		AL03_Kort02_DI04				AT %I*			:BOOL;	
		AL03_Kort02_DI05				AT %I*			:BOOL;	
		AL03_Kort02_DI06				AT %I*			:BOOL;	
		AL03_Kort02_DI07				AT %I*			:BOOL;	
		AL03_Kort02_DI08				AT %I*			:BOOL;	
										
										
	(* Digital Ut, KL2408 *)									
	(*Kort3*)									
		AL03_Kort03_DU01				AT %Q*			:BOOL;	
		AL03_Kort03_DU02				AT %Q*			:BOOL;	
		AL03_Kort03_DU03				AT %Q*			:BOOL;	
		AL03_Kort03_DU04				AT %Q*			:BOOL;	
		AL03_Kort03_DU05				AT %Q*			:BOOL;	
		AL03_Kort03_DU06				AT %Q*			:BOOL;	
		AL03_Kort03_DU07				AT %Q*			:BOOL;	
		AL03_Kort03_DU08				AT %Q*			:BOOL;
										
										
										


												

END_VAR

(* Global variable list: HUS3/AL03/HUS3_AL03_IO_Program *)
VAR_GLOBAL

					(*	Name	Device	Address	Data type	Rawmin	Rawmax	Engmin	Engmax	Unit	Format	Description	Alarmoptions	Trendoptions	*)		
	(* Digitala in, KL1488  *)																				
	(*Kort 1*)																				
		HUS3_AL03_FS01_L	AT%MX226.0	:BOOL;	(*	HUS3_AL03_FS01_L	AS01	GVL.HUS3_AL03_FS01_L	DIGITAL	0	0	0	0			Utlöst dvärgbrytare 	p:B		*)
		HUS3_LB05_HD75_L	AT%MX226.1	:BOOL;	(*	HUS3_LB05_HD75_L	AS01	GVL.HUS3_LB05_HD75_L	DIGITAL	0	0	0	0			Utlöst rökdetektor 	p:A		*)		
		HUS3_LB05_HD75_L1	AT%MX226.2	:BOOL;	(*	HUS3_LB05_HD75_L1	AS01	GVL.HUS3_LB05_HD75_L1	DIGITAL	0	0	0	0			Servicelarm	p:B		*)
		HUS3_LB05_HD75_L2	AT%MX226.3	:BOOL;	(*	HUS3_LB05_HD75_L2	AS01	GVL.HUS3_LB05_HD75_L2	DIGITAL	0	0	0	0			Fellarm 	p:B		*)
		HUS3_LB05_BS208_IO	AT%MX226.4	:BOOL;	(*	HUS3_LB05_BS208_IO	AS01	GVL.HUS3_LB05_BS208_IO	DIGITAL	0	0	0	0			Indikering öppet 			*)		
		HUS3_LB05_BS208_IS	AT%MX226.5	:BOOL;	(*	HUS3_LB05_BS208_IS	AS01	GVL.HUS3_LB05_BS208_IS	DIGITAL	0	0	0	0			Indikering stängt 			*)		
		HUS3_LB05_BS209_IO	AT%MX226.6	:BOOL;	(*	HUS3_LB05_BS209_IO	AS01	GVL.HUS3_LB05_BS209_IO	DIGITAL	0	0	0	0			Indikering öppet 			*)		
		HUS3_LB05_BS209_IS	AT%MX226.7	:BOOL;	(*	HUS3_LB05_BS209_IS	AS01	GVL.HUS3_LB05_BS209_IS	DIGITAL	0	0	0	0			Indikering stängt 			*)		
																					
																					
	(* Digitala in, KL1488  *)																				
	(*Kort 2*)																				
		HUS3_LB05_BS210_IO	AT%MX227.0	:BOOL;	(*	HUS3_LB05_BS210_IO	AS01	GVL.HUS3_LB05_BS210_IO	DIGITAL	0	0	0	0			Indikering öppet 	p:A		*)		
		HUS3_LB05_BS210_IS	AT%MX227.1	:BOOL;	(*	HUS3_LB05_BS210_IS	AS01	GVL.HUS3_LB05_BS210_IS	DIGITAL	0	0	0	0			Indikering stängt 	p:B		*)		
		HUS3_AL03_RESERV_DI_KORT02_CH03	AT%MX227.2	:BOOL;	(*											Reserv 			*)		
		HUS3_AL03_RESERV_DI_KORT02_CH04	AT%MX227.3	:BOOL;	(*											Reserv 			*)		
		HUS3_AL03_RESERV_DI_KORT02_CH05	AT%MX227.4	:BOOL;	(*											Reserv 			*)		
		HUS3_AL03_RESERV_DI_KORT02_CH06	AT%MX227.5	:BOOL;	(*											Reserv 			*)		
		HUS3_AL03_RESERV_DI_KORT02_CH07	AT%MX227.6	:BOOL;	(*											Reserv 			*)		
		HUS3_AL03_RESERV_DI_KORT02_CH08	AT%MX227.7	:BOOL;	(*											Reserv 			*)		
																					
																					
	(* Digital Ut, KL2408 *)																				
	(*Kort 3*)																				
		HUS3_LB05_BS208_M	AT%MX228.0	:BOOL;	(*											Manöver			*)		
		HUS3_LB05_BS209_M	AT%MX228.1	:BOOL;	(*											Manöver			*)		
		HUS3_LB05_BS210_M	AT%MX228.2	:BOOL;	(*											Manöver 			*)		
		HUS3_AL03_RESERV_DU_KORT03_CH04	AT%MX228.3	:BOOL;	(*											Reserv 			*)		
		HUS3_AL03_RESERV_DU_KORT03_CH05	AT%MX228.4	:BOOL;	(*											Reserv 			*)		
		HUS3_AL03_RESERV_DU_KORT03_CH06	AT%MX228.5	:BOOL;	(*											Reserv 			*)		
		HUS3_AL03_RESERV_DU_KORT03_CH07	AT%MX228.6	:BOOL;	(*											Reserv 			*)		
		HUS3_AL03_RESERV_DU_KORT03_CH08	AT%MX228.7	:BOOL;	(*											Reserv 			*)		
																					
																					


END_VAR

(* Global variable list: HUS3/AS03/HUS3_AS03_IO_Hardvara *)
VAR_GLOBAL


	(* Digitala in, KL1488  *)										
	(*Kort1*)										
		AS03_Kort01_DI01				AT %I*			:BOOL;		
		AS03_Kort01_DI02				AT %I*			:BOOL;		
		AS03_Kort01_DI03				AT %I*			:BOOL;		
		AS03_Kort01_DI04				AT %I*			:BOOL;		
		AS03_Kort01_DI05				AT %I*			:BOOL;		
		AS03_Kort01_DI06				AT %I*			:BOOL;		
		AS03_Kort01_DI07				AT %I*			:BOOL;		
		AS03_Kort01_DI08				AT %I*			:BOOL;		
											
											
	(* Digitala in, KL1488  *)										
	(*Kort2*)										
		AS03_Kort02_DI01				AT %I*			:BOOL;		
		AS03_Kort02_DI02				AT %I*			:BOOL;		
		AS03_Kort02_DI03				AT %I*			:BOOL;		
		AS03_Kort02_DI04				AT %I*			:BOOL;		
		AS03_Kort02_DI05				AT %I*			:BOOL;		
		AS03_Kort02_DI06				AT %I*			:BOOL;		
		AS03_Kort02_DI07				AT %I*			:BOOL;		
		AS03_Kort02_DI08				AT %I*			:BOOL;		
											
											
	(* Digital Ut, KL2408 *)
	(*Kort3*)										
		AS03_Kort03_DU01				AT %Q*			:BOOL;		
		AS03_Kort03_DU02				AT %Q*			:BOOL;		
		AS03_Kort03_DU03				AT %Q*			:BOOL;		
		AS03_Kort03_DU04				AT %Q*			:BOOL;		
		AS03_Kort03_DU05				AT %Q*			:BOOL;		
		AS03_Kort03_DU06				AT %Q*			:BOOL;		
		AS03_Kort03_DU07				AT %Q*			:BOOL;		
		AS03_Kort03_DU08				AT %Q*			:BOOL;		
											

(*	(* Analoga in, KL3208-0010, PT1000 *)										
	(*Kort5*)										
		AS03_Kort04_AI01									
		AS03_Kort04_AI02									
		AS03_Kort04_AI03									
		AS03_Kort04_AI04									
		AS03_Kort04_AI05									
		AS03_Kort04_AI06									
		AS03_Kort04_AI07									
		AS03_Kort04_AI08					*)				
											

	(* Analoga Ut, KL4408 *)								
	(*Kort5*)								
		AS03_Kort05_AU01				AT %Q*			:INT;
		AS03_Kort05_AU02				AT %Q*			:INT;
		AS03_Kort05_AU03				AT %Q*			:INT;
		AS03_Kort05_AU04				AT %Q*			:INT;
		AS03_Kort05_AU05				AT %Q*			:INT;
		AS03_Kort05_AU06				AT %Q*			:INT;
		AS03_Kort05_AU07				AT %Q*			:INT;
		AS03_Kort05_AU08				AT %Q*			:INT;
									
									



END_VAR

(* Global variable list: HUS3/AS03/HUS3_AS03_IO_Program *)
VAR_GLOBAL



					(*	Name	Device	Address	Data type	Rawmin	Rawmax	Engmin	Engmax	Unit	Format	Description	Alarmoptions	Trendoptions	*)	
	(* Digitala in, KL1488  *)																			
	(*Kort 1*)																			
		HUS3_AS03_FB01_L	AT%MX230.0	:BOOL;	(*	HUS3_AS03_FB01_L	AS01	GVL.HUS3_AS03_FB01_L	DIGITAL	0	0	0	0			Fasbrott/fel fasföljd	p:A		*)	
		HUS3_AS03_JFB01_L	AT%MX230.1	:BOOL;	(*	HUS3_AS03_JFB01_L	AS01	GVL.HUS3_AS03_JFB01_L	DIGITAL	0	0	0	0			Jordfelsbrytare 	p:B		*)	
		HUS3_AS03_FS01_L	AT%MX230.2	:BOOL;	(*	HUS3_AS03_FS01_L	AS01	GVL.HUS3_AS03_FS01_L	DIGITAL	0	0	0	0			Utlöst dvärgbrytare 	p:B		*)	
		HUS3_AS03_RESERV_DI_KORT01_CH04	AT%MX230.3	:BOOL;	(*											Reserv 			*)	
		HUS3_AS03_RESERV_DI_KORT01_CH05	AT%MX230.4	:BOOL;	(*											Reserv 			*)	
		HUS3_AS03_RESERV_DI_KORT01_CH06	AT%MX230.5	:BOOL;	(*											Reserv 			*)	
		HUS3_AS03_RESERV_DI_KORT01_CH07	AT%MX230.6	:BOOL;	(*											Reserv 			*)	
		HUS3_AS03_RESERV_DI_KORT01_CH08	AT%MX230.7	:BOOL;	(*											Reserv 			*)	
																				
																				
	(* Digitala in, KL1488  *)																			
	(*Kort 2*)																			
		HUS3_VS40_PV01_IT	AT%MX231.0	:BOOL;	(*	HUS3_VS40_PV01_IT	AS01	GVL.HUS3_VS40_PV01_IT	DIGITAL	0	0	0	0			Driftindikering cirkulationspump			*)	
		HUS3_FA301_FF01_LD	AT%MX231.1	:BOOL;	(*	HUS3_FA301_FF01_LD	AS01	GVL.HUS3_FA301_FF01_LD	DIGITAL	0	0	0	0			Driftfel frånluftsfläkt			*)	
		HUS3_FA302_FF01_LD	AT%MX231.2	:BOOL;	(*	HUS3_FA302_FF01_LD	AS01	GVL.HUS3_FA302_FF01_LD	DIGITAL	0	0	0	0			Driftfel frånluftsfläkt			*)	
		HUS3_FA303_FF01_LD	AT%MX231.3	:BOOL;	(*	HUS3_FA303_FF01_LD	AS01	GVL.HUS3_FA303_FF01_LD	DIGITAL	0	0	0	0			Driftfel frånluftsfläkt			*)	
		HUS3_AS03_RESERV_DI_KORT02_CH05	AT%MX231.4	:BOOL;	(*											Reserv 			*)	
		HUS3_AS03_RESERV_DI_KORT02_CH06	AT%MX231.5	:BOOL;	(*											Reserv 			*)	
		HUS3_AS03_RESERV_DI_KORT02_CH07	AT%MX231.6	:BOOL;	(*											Reserv 			*)	
		HUS3_AS03_RESERV_DI_KORT02_CH08	AT%MX231.7	:BOOL;	(*											Reserv 			*)	
																				
																				
	(* Digital Ut, KL2408 *)																			
	(*Kort 3*)																			
		HUS3_AS03_SA01_M	AT%MX232.0	:BOOL;	(*											Summalarm AS01 			*)
		HUS3_VS40_PV01_M	AT%MX232.1	:BOOL;	(*											Manöver			*)	
		HUS3_AS03_RESERV_DU_KORT03_CH03	AT%MX232.2	:BOOL;	(*											Reserv 			*)	
		HUS3_AS03_RESERV_DU_KORT03_CH04	AT%MX232.3	:BOOL;	(*											Reserv 			*)	
		HUS3_AS03_RESERV_DU_KORT03_CH05	AT%MX232.4	:BOOL;	(*											Reserv 			*)	
		HUS3_AS03_RESERV_DU_KORT03_CH06	AT%MX232.5	:BOOL;	(*											Reserv 			*)	
		HUS3_AS03_RESERV_DU_KORT03_CH07	AT%MX232.6	:BOOL;	(*											Reserv 			*)	
		HUS3_AS03_RESERV_DU_KORT03_CH08	AT%MX232.7	:BOOL;	(*											Reserv 			*)	
																				
																				
	(* Analoga in, KL3208-0010, PT1000  *)																			
	(*Kort 4*)																			
		HUS3_VS40_GT11_MV	AT%MB236	:REAL;	(*	HUS3_VS40_GT11_MV	AS01	GVL.HUS3_VS40_GT11_MV	REAL	-50	150	-50	150	°C	0.0	Mätvärde tilloppstemperatur			*)	
		HUS3_VS40_GT41_MV	AT%MB240	:REAL;	(*	HUS3_VS40_GT41_MV	AS01	GVL.HUS3_VS40_GT41_MV	REAL	-50	150	-50	150	°C	0.0	Mätvärde returtemperatur			*)	
		HUS3_FA301_GT51_MV	AT%MB244	:REAL;	(*	HUS3_FA301_GT51_MV	AS01	GVL.HUS3_FA301_GT51_MV	REAL	-50	150	-50	150	°C	0.0	Mätvärde frånluftstemperatur			*)	
		HUS3_FA302_GT51_MV	AT%MB248	:REAL;	(*	HUS3_FA302_GT51_MV	AS01	GVL.HUS3_FA302_GT51_MV	REAL	-50	150	-50	150	°C	0.0	Mätvärde frånluftstemperatur			*)	
		HUS3_FA303_GT51_MV	AT%MB252	:REAL;	(*	HUS3_FA303_GT51_MV	AS01	GVL.HUS3_FA303_GT51_MV	REAL	-50	150	-50	150	°C	0.0	Mätvärde frånluftstemperatur			*)
		HUS3_AS03_RESERV_AI_KORT04_CH06	AT%MB256	:REAL;	(*											Reserv			*)
		HUS3_AS03_RESERV_AI_KORT04_CH07	AT%MB260	:REAL;	(*											Reserv			*)
		HUS3_AS03_RESERV_AI_KORT04_CH08	AT%MB264	:REAL;	(*											Reserv			*)
																				
																				
	(* Analoga ut, KL4408  *)																			
	(*Kort 5*)																			
		HUS3_VS40_SV21_R	AT%MB268	:REAL;	(*	HUS3_VS40_SV21_R	AS01	GVL.HUS3_VS40_SV21_R	REAL	0	100	0	100	%		Styrsignal ventilställdon			*)	
		HUS3_FA301_FF01_R	AT%MB272	:REAL;	(*	HUS3_FA301_FF01_R	AS01	GVL.HUS3_FA301_FF01_R	REAL	0	100	0	100	%		Styrsignal frånluftsfläkt			*)	
		HUS3_FA302_FF01_R	AT%MB276	:REAL;	(*	HUS3_FA302_FF01_R	AS01	GVL.HUS3_FA302_FF01_R	REAL	0	100	0	100	%		Styrsignal frånluftsfläkt			*)	
		HUS3_FA303_FF01_R	AT%MB280	:REAL;	(*	HUS3_FA303_FF01_R	AS01	GVL.HUS3_FA303_FF01_R	REAL	0	100	0	100	%		Styrsignal frånluftsfläkt			*)	
		HUS3_AS03_RESERV_AU_KORT05_CH05	AT%MB284	:REAL;	(*											Reserv			*)	
		HUS3_AS03_RESERV_AU_KORT05_CH06	AT%MB288	:REAL;	(*											Reserv			*)	
		HUS3_AS03_RESERV_AU_KORT05_CH07	AT%MB292	:REAL;	(*											Reserv			*)	
		HUS3_AS03_RESERV_AU_KORT05_CH08	AT%MB296	:REAL;	(*											Reserv			*)	
																				
																				
																				
																				
																				
																				
																				
																				

											


END_VAR

(* Global variable list: HUS2/BS205, BS206, BS207/HUS3_BS205_207_INST *)
VAR_GLOBAL PERSISTENT


																		
				(*	Name	Device	Address	Data type	Rawmin	Rawmax	Engmin	Engmax	Unit	Format	Description	Alarmoptions	Trendoptions	*)
																		
																		
																		
																		
																		
	HUS3_LB04_BS205_MAN	AT%MB3540	:INT;	(*	HUS3_LB04_BS205_MAN	AS01	GVL.HUS3_LB04_BS205_MAN	INT	0	2	0	2			Manuell styrning brandspjäll 0=Auto,1=Från,2=Till			*)
	HUS3_LB04_BS205_FLM	AT%MB3542	:INT;	(*	HUS3_LB04_BS205_FLM	AS01	GVL.HUS3_LB04_BS205_FLM	INT	0	3600	0	3600	Min		Larmfördröjning brandspjäll ej i AUTO			*)
	HUS3_LB04_BS205_FL	AT%MB3544	:INT;	(*	HUS3_LB04_BS205_FL	AS01	GVL.HUS3_LB04_BS205_FL	INT	0	1000	0	1000	Sek		Larmfördröjning brandspjäll öppnar ej			*)
	HUS3_LB04_BS205_FL1	AT%MB3546	:INT;	(*	HUS3_LB04_BS205_FL1	AS01	GVL.HUS3_LB04_BS205_FL1	INT	0	1000	0	1000	Sek		Larmfördröjning brandspjäll stänger ej			*)
	HUS3_LB04_BS206_MAN	AT%MB3548	:INT;	(*	HUS3_LB04_BS206_MAN	AS01	GVL.HUS3_LB04_BS206_MAN	INT	0	2	0	2			Manuell styrning brandspjäll 0=Auto,1=Från,2=Till			*)
	HUS3_LB04_BS206_FLM	AT%MB3550	:INT;	(*	HUS3_LB04_BS206_FLM	AS01	GVL.HUS3_LB04_BS206_FLM	INT	0	3600	0	3600	Min		Larmfördröjning brandspjäll ej i AUTO			*)
	HUS3_LB04_BS206_FL	AT%MB3552	:INT;	(*	HUS3_LB04_BS206_FL	AS01	GVL.HUS3_LB04_BS206_FL	INT	0	1000	0	1000	Sek		Larmfördröjning brandspjäll öppnar ej			*)
	HUS3_LB04_BS206_FL1	AT%MB3554	:INT;	(*	HUS3_LB04_BS206_FL1	AS01	GVL.HUS3_LB04_BS206_FL1	INT	0	1000	0	1000	Sek		Larmfördröjning brandspjäll stänger ej			*)
	HUS3_LB04_BS207_MAN	AT%MB3556	:INT;	(*	HUS3_LB04_BS207_MAN	AS01	GVL.HUS3_LB04_BS207_MAN	INT	0	2	0	2			Manuell styrning brandspjäll 0=Auto,1=Från,2=Till			*)
	HUS3_LB04_BS207_FLM	AT%MB3558	:INT;	(*	HUS3_LB04_BS207_FLM	AS01	GVL.HUS3_LB04_BS207_FLM	INT	0	3600	0	3600	Min		Larmfördröjning brandspjäll ej i AUTO			*)
	HUS3_LB04_BS207_FL	AT%MB3560	:INT;	(*	HUS3_LB04_BS207_FL	AS01	GVL.HUS3_LB04_BS207_FL	INT	0	1000	0	1000	Sek		Larmfördröjning brandspjäll öppnar ej			*)
	HUS3_LB04_BS207_FL1	AT%MB3562	:INT;	(*	HUS3_LB04_BS207_FL1	AS01	GVL.HUS3_LB04_BS207_FL1	INT	0	1000	0	1000	Sek		Larmfördröjning brandspjäll stänger ej			*)
																		
																		
																		
																		



END_VAR
																
																

(* Global variable list: HUS2/BS205, BS206, BS207/HUS3_BS205_207_LARM *)
VAR_GLOBAL


																			
																			
																			
		HUS3_LB04_BS205_LM	AT%MX3600.0	:BOOL; 	(*	HUS3_LB04_BS205_LM	AS01	GVL.HUS3_LB04_BS205_LM	DIGITAL	0	0	0	0			Brandspjäll ej i läge AUTO	p:C		*)
		HUS3_LB04_BS205_L	AT%MX3600.1	:BOOL; 	(*	HUS3_LB04_BS205_L	AS01	GVL.HUS3_LB04_BS205_L	DIGITAL	0	0	0	0			Brandspjäll öppnar ej	p:B		*)
		HUS3_LB04_BS205_L1	AT%MX3600.2	:BOOL; 	(*	HUS3_LB04_BS205_L1	AS01	GVL.HUS3_LB04_BS205_L1	DIGITAL	0	0	0	0			Brandspjäll stänger ej	p:B		*)
		HUS3_LB04_BS205_L2	AT%MX3600.3	:BOOL; 	(*	HUS3_LB04_BS205_L2	AS01	GVL.HUS3_LB04_BS205_L2	DIGITAL	0	0	0	0			Brandspjäll stängt och öppet samtidigt	p:B		*)
		HUS3_LB04_BS205_ACK	AT%MX3600.4	:BOOL; 	(*	HUS3_LB04_BS205_ACK	AS01	GVL.HUS3_LB04_BS205_ACK	DIGITAL	0	0	0	0			Larmkvittens brandspjäll BS205			*)
		HUS3_LB04_BS206_LM	AT%MX3600.5	:BOOL; 	(*	HUS3_LB04_BS206_LM	AS01	GVL.HUS3_LB04_BS206_LM	DIGITAL	0	0	0	0			Brandspjäll ej i läge AUTO	p:C		*)
		HUS3_LB04_BS206_L	AT%MX3600.6	:BOOL; 	(*	HUS3_LB04_BS206_L	AS01	GVL.HUS3_LB04_BS206_L	DIGITAL	0	0	0	0			Brandspjäll öppnar ej	p:B		*)
		HUS3_LB04_BS206_L1	AT%MX3600.7	:BOOL; 	(*	HUS3_LB04_BS206_L1	AS01	GVL.HUS3_LB04_BS206_L1	DIGITAL	0	0	0	0			Brandspjäll stänger ej	p:B		*)
		HUS3_LB04_BS206_L2	AT%MX3601.0	:BOOL; 	(*	HUS3_LB04_BS206_L2	AS01	GVL.HUS3_LB04_BS206_L2	DIGITAL	0	0	0	0			Brandspjäll stängt och öppet samtidigt	p:B		*)
		HUS3_LB04_BS206_ACK	AT%MX3601.1	:BOOL; 	(*	HUS3_LB04_BS206_ACK	AS01	GVL.HUS3_LB04_BS206_ACK	DIGITAL	0	0	0	0			Larmkvittens brandspjäll BS206			*)
		HUS3_LB04_BS207_LM	AT%MX3601.2	:BOOL; 	(*	HUS3_LB04_BS207_LM	AS01	GVL.HUS3_LB04_BS207_LM	DIGITAL	0	0	0	0			Brandspjäll ej i läge AUTO	p:C		*)
		HUS3_LB04_BS207_L	AT%MX3601.3	:BOOL; 	(*	HUS3_LB04_BS207_L	AS01	GVL.HUS3_LB04_BS207_L	DIGITAL	0	0	0	0			Brandspjäll öppnar ej	p:B		*)
		HUS3_LB04_BS207_L1	AT%MX3601.4	:BOOL; 	(*	HUS3_LB04_BS207_L1	AS01	GVL.HUS3_LB04_BS207_L1	DIGITAL	0	0	0	0			Brandspjäll stänger ej	p:B		*)
		HUS3_LB04_BS207_L2	AT%MX3601.5	:BOOL; 	(*	HUS3_LB04_BS207_L2	AS01	GVL.HUS3_LB04_BS207_L2	DIGITAL	0	0	0	0			Brandspjäll stängt och öppet samtidigt	p:B		*)
		HUS3_LB04_BS207_ACK	AT%MX3601.6	:BOOL; 	(*	HUS3_LB04_BS207_ACK	AS01	GVL.HUS3_LB04_BS207_ACK	DIGITAL	0	0	0	0			Larmkvittens brandspjäll BS207			*)
																			
																			
																			
																			
																			
																			
																			
																			


END_VAR

(* Global variable list: HUS2/BS205, BS206, BS207/HUS3_BS205_207_OVRIGT *)
VAR_GLOBAL


	HUS3_LB04_BS205_IT	AT%MX3604.0	:BOOL;	(*	HUS3_LB04_BS205_IT	AS01	GVL.HUS3_LB04_BS205_IT	DIGITAL	0	0	0	0			Motionering aktiv			*)
	HUS3_LB04_BS206_IT	AT%MX3604.1	:BOOL;	(*	HUS3_LB04_BS206_IT	AS01	GVL.HUS3_LB04_BS206_IT	DIGITAL	0	0	0	0			Motionering aktiv			*)
	HUS3_LB04_BS207_IT	AT%MX3604.2	:BOOL;	(*	HUS3_LB04_BS207_IT	AS01	GVL.HUS3_LB04_BS207_IT	DIGITAL	0	0	0	0			Motionering aktiv			*)
																						


END_VAR

(* Global variable list: HUS3/BS208, BS209, BS210/HUS3_BS208_210_INST *)
VAR_GLOBAL PERSISTENT

				(*	Name	Device	Address	Data type	Rawmin	Rawmax	Engmin	Engmax	Unit	Format	Description	Alarmoptions	Trendoptions	*)


																		
	HUS3_LB05_BS208_MAN	AT%MB3610	:INT;	(*	HUS3_LB05_BS208_MAN	AS01	GVL.HUS3_LB05_BS208_MAN	INT	0	2	0	2			Manuell styrning brandspjäll 0=Auto,1=Från,2=Till			*)
	HUS3_LB05_BS208_FLM	AT%MB3612	:INT;	(*	HUS3_LB05_BS208_FLM	AS01	GVL.HUS3_LB05_BS208_FLM	INT	0	3600	0	3600	Min		Larmfördröjning brandspjäll ej i AUTO			*)
	HUS3_LB05_BS208_FL	AT%MB3614	:INT;	(*	HUS3_LB05_BS208_FL	AS01	GVL.HUS3_LB05_BS208_FL	INT	0	1000	0	1000	Sek		Larmfördröjning brandspjäll öppnar ej			*)
	HUS3_LB05_BS208_FL1	AT%MB3616	:INT;	(*	HUS3_LB05_BS208_FL1	AS01	GVL.HUS3_LB05_BS208_FL1	INT	0	1000	0	1000	Sek		Larmfördröjning brandspjäll stänger ej			*)
	HUS3_LB05_BS209_MAN	AT%MB3618	:INT;	(*	HUS3_LB05_BS209_MAN	AS01	GVL.HUS3_LB05_BS209_MAN	INT	0	2	0	2			Manuell styrning brandspjäll 0=Auto,1=Från,2=Till			*)
	HUS3_LB05_BS209_FLM	AT%MB3620	:INT;	(*	HUS3_LB05_BS209_FLM	AS01	GVL.HUS3_LB05_BS209_FLM	INT	0	3600	0	3600	Min		Larmfördröjning brandspjäll ej i AUTO			*)
	HUS3_LB05_BS209_FL	AT%MB3622	:INT;	(*	HUS3_LB05_BS209_FL	AS01	GVL.HUS3_LB05_BS209_FL	INT	0	1000	0	1000	Sek		Larmfördröjning brandspjäll öppnar ej			*)
	HUS3_LB05_BS209_FL1	AT%MB3624	:INT;	(*	HUS3_LB05_BS209_FL1	AS01	GVL.HUS3_LB05_BS209_FL1	INT	0	1000	0	1000	Sek		Larmfördröjning brandspjäll stänger ej			*)
	HUS3_LB05_BS210_MAN	AT%MB3626	:INT;	(*	HUS3_LB05_BS210_MAN	AS01	GVL.HUS3_LB05_BS210_MAN	INT	0	2	0	2			Manuell styrning brandspjäll 0=Auto,1=Från,2=Till			*)
	HUS3_LB05_BS210_FLM	AT%MB3628	:INT;	(*	HUS3_LB05_BS210_FLM	AS01	GVL.HUS3_LB05_BS210_FLM	INT	0	3600	0	3600	Min		Larmfördröjning brandspjäll ej i AUTO			*)
	HUS3_LB05_BS210_FL	AT%MB3630	:INT;	(*	HUS3_LB05_BS210_FL	AS01	GVL.HUS3_LB05_BS210_FL	INT	0	1000	0	1000	Sek		Larmfördröjning brandspjäll öppnar ej			*)
	HUS3_LB05_BS210_FL1	AT%MB3632	:INT;	(*	HUS3_LB05_BS210_FL1	AS01	GVL.HUS3_LB05_BS210_FL1	INT	0	1000	0	1000	Sek		Larmfördröjning brandspjäll stänger ej			*)
																		


END_VAR

																

(* Global variable list: HUS3/BS208, BS209, BS210/HUS3_BS208_210_LARM *)
VAR_GLOBAL


		HUS3_LB05_BS208_LM	AT%MX3670.0	:BOOL; 	(*	HUS3_LB05_BS208_LM	AS01	GVL.HUS3_LB05_BS208_LM	DIGITAL	0	0	0	0			Brandspjäll ej i läge AUTO	p:C		*)		
		HUS3_LB05_BS208_L	AT%MX3670.1	:BOOL; 	(*	HUS3_LB05_BS208_L	AS01	GVL.HUS3_LB05_BS208_L	DIGITAL	0	0	0	0			Brandspjäll öppnar ej	p:B		*)
		HUS3_LB05_BS208_L1	AT%MX3670.2	:BOOL; 	(*	HUS3_LB05_BS208_L1	AS01	GVL.HUS3_LB05_BS208_L1	DIGITAL	0	0	0	0			Brandspjäll stänger ej	p:B		*)		
		HUS3_LB05_BS208_L2	AT%MX3670.3	:BOOL; 	(*	HUS3_LB05_BS208_L2	AS01	GVL.HUS3_LB05_BS208_L2	DIGITAL	0	0	0	0			Brandspjäll stängt och öppet samtidigt	p:B		*)		
		HUS3_LB05_BS208_ACK	AT%MX3670.4	:BOOL; 	(*	HUS3_LB05_BS208_ACK	AS01	GVL.HUS3_LB05_BS208_ACK	DIGITAL	0	0	0	0			Larmkvittens brandspjäll BS208			*)		
		HUS3_LB05_BS209_LM	AT%MX3670.5	:BOOL; 	(*	HUS3_LB05_BS209_LM	AS01	GVL.HUS3_LB05_BS209_LM	DIGITAL	0	0	0	0			Brandspjäll ej i läge AUTO	p:C		*)		
		HUS3_LB05_BS209_L	AT%MX3670.6	:BOOL; 	(*	HUS3_LB05_BS209_L	AS01	GVL.HUS3_LB05_BS209_L	DIGITAL	0	0	0	0			Brandspjäll öppnar ej	p:B		*)		
		HUS3_LB05_BS209_L1	AT%MX3670.7	:BOOL; 	(*	HUS3_LB05_BS209_L1	AS01	GVL.HUS3_LB05_BS209_L1	DIGITAL	0	0	0	0			Brandspjäll stänger ej	p:B		*)		
		HUS3_LB05_BS209_L2	AT%MX3671.0	:BOOL; 	(*	HUS3_LB05_BS209_L2	AS01	GVL.HUS3_LB05_BS209_L2	DIGITAL	0	0	0	0			Brandspjäll stängt och öppet samtidigt	p:B		*)		
		HUS3_LB05_BS209_ACK	AT%MX3671.1	:BOOL; 	(*	HUS3_LB05_BS209_ACK	AS01	GVL.HUS3_LB05_BS209_ACK	DIGITAL	0	0	0	0			Larmkvittens brandspjäll BS209			*)		
		HUS3_LB05_BS210_LM	AT%MX3671.2	:BOOL; 	(*	HUS3_LB05_BS210_LM	AS01	GVL.HUS3_LB05_BS210_LM	DIGITAL	0	0	0	0			Brandspjäll ej i läge AUTO	p:C		*)		
		HUS3_LB05_BS210_L	AT%MX3671.3	:BOOL; 	(*	HUS3_LB05_BS210_L	AS01	GVL.HUS3_LB05_BS210_L	DIGITAL	0	0	0	0			Brandspjäll öppnar ej	p:B		*)		
		HUS3_LB05_BS210_L1	AT%MX3671.4	:BOOL; 	(*	HUS3_LB05_BS210_L1	AS01	GVL.HUS3_LB05_BS210_L1	DIGITAL	0	0	0	0			Brandspjäll stänger ej	p:B		*)		
		HUS3_LB05_BS210_L2	AT%MX3671.5	:BOOL; 	(*	HUS3_LB05_BS210_L2	AS01	GVL.HUS3_LB05_BS210_L2	DIGITAL	0	0	0	0			Brandspjäll stängt och öppet samtidigt	p:B		*)		
		HUS3_LB05_BS210_ACK	AT%MX3671.6	:BOOL; 	(*	HUS3_LB05_BS210_ACK	AS01	GVL.HUS3_LB05_BS210_ACK	DIGITAL	0	0	0	0			Larmkvittens brandspjäll BS210			*)		
																					
																					


END_VAR

(* Global variable list: HUS3/BS208, BS209, BS210/HUS3_BS208_210_OVRIGT *)
VAR_GLOBAL

																							
		HUS3_LB05_BS208_IT	AT%MX3674.0	:BOOL;	(*	HUS3_LB05_BS208_IT	AS01	GVL.HUS3_LB05_BS208_IT	DIGITAL	0	0	0	0			Motionering aktiv			*)
		HUS3_LB05_BS209_IT	AT%MX3674.1	:BOOL;	(*	HUS3_LB05_BS209_IT	AS01	GVL.HUS3_LB05_BS209_IT	DIGITAL	0	0	0	0			Motionering aktiv			*)
		HUS3_LB05_BS210_IT	AT%MX3674.2	:BOOL;	(*	HUS3_LB05_BS210_IT	AS01	GVL.HUS3_LB05_BS210_IT	DIGITAL	0	0	0	0			Motionering aktiv			*)
																							


END_VAR

(* Global variable list: HUS3/FA301, FA302, FA303/HUS3_FA301_303_INST *)
VAR_GLOBAL PERSISTENT

																			

																			
					(*	Name	Device	Address	Data type	Rawmin	Rawmax	Engmin	Engmax	Unit	Format	Description	Alarmoptions	Trendoptions	*)
																			
		HUS3_FA301_SO1_MAN	AT%MB4000	:INT;	(*	HUS3_FA301_SO1_MAN	AS01	GVL.HUS3_FA301_SO1_MAN	INT	0	2	0	2			Manuell styrning system FA301. 0=Auto, 1=Manuell från, 2=Manuell till			*)
		HUS3_FA301_SO1_FLM	AT%MB4002	:INT;	(*	HUS3_FA301_SO1_FLM	AS01	GVL.HUS3_FA301_SO1_FLM	INT	0	3600	0	3600	Min		Larmfördröjning serviceomkopplare ej i läge AUTO			*)
																			
		HUS3_FA301_FF01_FLM	AT%MB4004	:INT;	(*	HUS3_FA301_FF01_FLM	AS01	GVL.HUS3_FA301_FF01_FLM	INT	0	3600	0	3600	Min		Larmfördröjning frånluftsfläkt ej i AUTO			*)
		HUS3_FA301_FF01_FLD	AT%MB4006	:INT;	(*	HUS3_FA301_FF01_FLD	AS01	GVL.HUS3_FA301_FF01_FLD	INT	0	120	0	120	Sek		Larmfördröjning driftfel frånluftsfläkt			*)
																			
		HUS3_FA301_FF01_MAN	AT%MB4008	:INT;	(*	HUS3_FA301_FF01_MAN	AS01	GVL.HUS3_FA301_FF01_MAN	INT	0	2	0	2			Manuell styrning frånluftsfläkt 0=Auto,1=Från,2=Till			*)
		HUS3_FA301_FF01_MAN1	AT%MB4010	:INT;	(*	HUS3_FA301_FF01_MAN	AS01	GVL.HUS3_FA301_FF01_MAN	INT	0	1	0	1			Manuell styrning styrsignal frånluftsfläkt 0=Auto,1=Till			*)
		HUS3_FA301_FF01_RMAN	AT%MB4012	:REAL;	(*	HUS3_FA301_FF01_RMAN	AS01	GVL.HUS3_FA301_FF01_RMAN	REAL	0	100	0	100	%		Manuell styrsignal frånluftsfläkt			*)
																			
		HUS3_FA301_GT51_STAG	AT%MB4016	:REAL;	(*	HUS3_FA301_GT51_STAG	AS01	GVL.HUS3_FA301_GT51_STAG	REAL	0	50	0	50	°C	0.0	Gränsvärde start forcering frånluftsfläkt			*)
		HUS3_FA301_GT51_STOG	AT%MB4020	:REAL;	(*	HUS3_FA301_GT51_STOG	AS01	GVL.HUS3_FA301_GT51_STOG	REAL	0	50	0	50	°C	0.0	Gränsvärde stopp forcering frånluftsfläkt			*)

		HUS3_FA301_GT51_GVH	AT%MB4024	:REAL;	(*	HUS3_FA301_GT51_GV	AS01	GVL.HUS3_FA301_GT51_GV	REAL	0	50	0	50	°C	0.0	Gränsvärde hög temperatur			*)
		HUS3_FA301_GT51_FLG	AT%MB4028	:INT;	(*	HUS3_FA301_GT51_FLG	AS01	GVL.HUS3_FA301_GT51_FLG	INT	0	3600	0	3600	Min		Lamfördröjning hög temperatur			*)
																			
																			
		HUS3_FA301_GT51_KRV	AT%MB4036	:REAL;	(*	HUS3_FA301_GT51_KRV	AS01	GVL.HUS3_FA301_GT51_KRV	REAL	-10	10	-10	10	°C	0.0	Kalibreringsvärde frånluftsgivare			*)
																			
		HUS3_FA301_FF01_BV	AT%MB4040	:REAL;	(*	HUS3_FA301_FF01_BV	AS01	GVL.HUS3_FA301_FF01_BV	REAL	0	100	0	100	%		Grundflöde frånluftsfläkt			*)
		HUS3_FA301_FF01_BV1	AT%MB4044	:REAL;	(*	HUS3_FA301_FF01_BV1	AS01	GVL.HUS3_FA301_FF01_BV1	REAL	0	100	0	100	%		Forcerat flöde frånluftsfläkt			*)
																			
																			
																			
																			
																			
																			
		HUS3_FA302_SO1_MAN	AT%MB4060	:INT;	(*	HUS3_FA302_SO1_MAN	AS01	GVL.HUS3_FA302_SO1_MAN	INT	0	2	0	2			Manuell styrning system FA302. 0=Auto, 1=Manuell från, 2=Manuell till			*)
		HUS3_FA302_SO1_FLM	AT%MB4062	:INT;	(*	HUS3_FA302_SO1_FLM	AS01	GVL.HUS3_FA302_SO1_FLM	INT	0	3600	0	3600	Min		Larmfördröjning serviceomkopplare ej i läge AUTO			*)
																			
		HUS3_FA302_FF01_FLM	AT%MB4064	:INT;	(*	HUS3_FA302_FF01_FLM	AS01	GVL.HUS3_FA302_FF01_FLM	INT	0	3600	0	3600	Min		Larmfördröjning frånluftsfläkt ej i AUTO			*)
		HUS3_FA302_FF01_FLD	AT%MB4066	:INT;	(*	HUS3_FA302_FF01_FLD	AS01	GVL.HUS3_FA302_FF01_FLD	INT	0	120	0	120	Sek		Larmfördröjning driftfel frånluftsfläkt			*)
																			
		HUS3_FA302_FF01_MAN	AT%MB4068	:INT;	(*	HUS3_FA302_FF01_MAN	AS01	GVL.HUS3_FA302_FF01_MAN	INT	0	2	0	2			Manuell styrning frånluftsfläkt 0=Auto,1=Från,2=Till			*)
		HUS3_FA302_FF01_MAN1	AT%MB4070	:INT;	(*	HUS3_FA302_FF01_MAN	AS01	GVL.HUS3_FA302_FF01_MAN	INT	0	1	0	1			Manuell styrning styrsignal frånluftsfläkt 0=Auto,1=Till			*)
		HUS3_FA302_FF01_RMAN	AT%MB4072	:REAL;	(*	HUS3_FA302_FF01_RMAN	AS01	GVL.HUS3_FA302_FF01_RMAN	REAL	0	100	0	100	%		Manuell styrsignal frånluftsfläkt			*)
																			
		HUS3_FA302_GT51_STAG	AT%MB4076	:REAL;	(*	HUS3_FA302_GT51_STAG	AS01	GVL.HUS3_FA302_GT51_STAG	REAL	0	50	0	50	°C	0.0	Gränsvärde start forcering frånluftsfläkt			*)
		HUS3_FA302_GT51_STOG	AT%MB4080	:REAL;	(*	HUS3_FA302_GT51_STOG	AS01	GVL.HUS3_FA302_GT51_STOG	REAL	0	50	0	50	°C	0.0	Gränsvärde stopp forcering frånluftsfläkt			*)

		HUS3_FA302_GT51_GVH	AT%MB4084	:REAL;	(*	HUS3_FA302_GT51_GV	AS01	GVL.HUS3_FA302_GT51_GV	REAL	0	50	0	50	°C	0.0	Gränsvärde hög temperatur			*)
		HUS3_FA302_GT51_FLG	AT%MB4088	:INT;	(*	HUS3_FA302_GT51_FLG	AS01	GVL.HUS3_FA302_GT51_FLG	INT	0	3600	0	3600	Min		Lamfördröjning hög temperatur			*)

																			
		HUS3_FA302_GT51_KRV	AT%MB4096	:REAL;	(*	HUS3_FA302_GT51_KRV	AS01	GVL.HUS3_FA302_GT51_KRV	REAL	-10	10	-10	10	°C	0.0	Kalibreringsvärde frånluftsgivare			*)
																			
		HUS3_FA302_FF01_BV	AT%MB4100	:REAL;	(*	HUS3_FA302_FF01_BV	AS01	GVL.HUS3_FA302_FF01_BV	REAL	0	100	0	100	%		Grundflöde frånluftsfläkt			*)
		HUS3_FA302_FF01_BV1	AT%MB4104	:REAL;	(*	HUS3_FA302_FF01_BV1	AS01	GVL.HUS3_FA302_FF01_BV1	REAL	0	100	0	100	%		Forcerat flöde frånluftsfläkt			*)
																			
																			
																			
																			
																			
																			
		HUS3_FA303_SO1_MAN	AT%MB4120	:INT;	(*	HUS3_FA303_SO1_MAN	AS01	GVL.HUS3_FA303_SO1_MAN	INT	0	2	0	2			Manuell styrning system FA303. 0=Auto, 1=Manuell från, 2=Manuell till			*)
		HUS3_FA303_SO1_FLM	AT%MB4122	:INT;	(*	HUS3_FA303_SO1_FLM	AS01	GVL.HUS3_FA303_SO1_FLM	INT	0	3600	0	3600	Min		Larmfördröjning serviceomkopplare ej i läge AUTO			*)
																			
		HUS3_FA303_FF01_FLM	AT%MB4124	:INT;	(*	HUS3_FA303_FF01_FLM	AS01	GVL.HUS3_FA303_FF01_FLM	INT	0	3600	0	3600	Min		Larmfördröjning frånluftsfläkt ej i AUTO			*)
		HUS3_FA303_FF01_FLD	AT%MB4126	:INT;	(*	HUS3_FA303_FF01_FLD	AS01	GVL.HUS3_FA303_FF01_FLD	INT	0	120	0	120	Sek		Larmfördröjning driftfel frånluftsfläkt			*)
																			
		HUS3_FA303_FF01_MAN	AT%MB4128	:INT;	(*	HUS3_FA303_FF01_MAN	AS01	GVL.HUS3_FA303_FF01_MAN	INT	0	2	0	2			Manuell styrning frånluftsfläkt 0=Auto,1=Från,2=Till			*)
		HUS3_FA303_FF01_MAN1	AT%MB4130	:INT;	(*	HUS3_FA303_FF01_MAN	AS01	GVL.HUS3_FA303_FF01_MAN	INT	0	1	0	1			Manuell styrning styrsignal frånluftsfläkt 0=Auto,1=Till			*)
		HUS3_FA303_FF01_RMAN	AT%MB4132	:REAL;	(*	HUS3_FA303_FF01_RMAN	AS01	GVL.HUS3_FA303_FF01_RMAN	REAL	0	100	0	100	%		Manuell styrsignal frånluftsfläkt			*)

		HUS3_FA303_GT51_STAG	AT%MB4136	:REAL;	(*	HUS3_FA303_GT51_STAG	AS01	GVL.HUS3_FA303_GT51_STAG	REAL	0	50	0	50	°C	0.0	Gränsvärde start forcering frånluftsfläkt			*)
		HUS3_FA303_GT51_STOG	AT%MB4140	:REAL;	(*	HUS3_FA303_GT51_STOG	AS01	GVL.HUS3_FA303_GT51_STOG	REAL	0	50	0	50	°C	0.0	Gränsvärde stopp forcering frånluftsfläkt			*)
																			
		HUS3_FA303_GT51_GVH	AT%MB4144	:REAL;	(*	HUS3_FA303_GT51_GVH	AS01	GVL.HUS3_FA303_GT51_GVH	REAL	0	50	0	50	°C	0.0	Gränsvärde hög temperatur			*)
		HUS3_FA303_GT51_FLG	AT%MB4148	:INT;	(*	HUS3_FA303_GT51_FLG	AS01	GVL.HUS3_FA303_GT51_FLG	INT	0	3600	0	3600	Min		Lamfördröjning hög temperatur			*)
																			
																			
		HUS3_FA303_GT51_KRV	AT%MB4156	:REAL;	(*	HUS3_FA303_GT51_KRV	AS01	GVL.HUS3_FA303_GT51_KRV	REAL	-10	10	-10	10	°C	0.0	Kalibreringsvärde frånluftsgivare			*)
																			
		HUS3_FA303_FF01_BV	AT%MB4160	:REAL;	(*	HUS3_FA303_FF01_BV	AS01	GVL.HUS3_FA303_FF01_BV	REAL	0	100	0	100	%		Grundflöde frånluftsfläkt			*)
		HUS3_FA303_FF01_BV1	AT%MB4164	:REAL;	(*	HUS3_FA303_FF01_BV1	AS01	GVL.HUS3_FA303_FF01_BV1	REAL	0	100	0	100	%		Forcerat flöde frånluftsfläkt			*)
																			
																			
																			
																			
																			
																			
																			
																			
																			
																			
																			
																			



END_VAR
																
																

(* Global variable list: HUS3/FA301, FA302, FA303/HUS3_FA301_303_LARM *)
VAR_GLOBAL



																			
																			
	HUS3_FA301_SO1_LM	AT%MX4200.0	:BOOL; 	(*	HUS3_FA301_SO1_LM	AS01	GVL.HUS3_FA301_SO1_LM	DIGITAL	0	0	0	0			Serviceomkopplare ej i läge AUTO	p:C		*)	
	HUS3_FA301_FF01_LM	AT%MX4200.1	:BOOL; 	(*	HUS3_FA301_FF01_LM	AS01	GVL.HUS3_FA301_FF01_LM	DIGITAL	0	0	0	0			Frånluftsfläkt ej i AUTO	p:B		*)	
	HUS3_FA301_GT51_LG	AT%MX4200.2	:BOOL; 	(*	HUS3_FA301_GT51_LG	AS01	GVL.HUS3_FA301_GT51_LG	DIGITAL	0	0	0	0			Givarfel frånluftsgivare	p:B		*)	
	HUS3_FA301_GT51_LH	AT%MX4200.3	:BOOL; 	(*	HUS3_FA301_GT51_LH	AS01	GVL.HUS3_FA301_GT51_LH	DIGITAL	0	0	0	0			Hög temperatur	p:B		*)	
																			
	HUS3_FA301_FF01_ACK	AT%MX4201.0	:BOOL; 	(*	HUS3_FA301_FF01_ACK	AS01	GVL.HUS3_FA301_FF01_ACK	DIGITAL	0	0	0	0			Larmkvittens frånluftsfläkt			*)
																			
																			
	HUS3_FA302_SO1_LM	AT%MX4202.0	:BOOL; 	(*	HUS3_FA302_SO1_LM	AS01	GVL.HUS3_FA302_SO1_LM	DIGITAL	0	0	0	0			Serviceomkopplare ej i läge AUTO	p:C		*)	
	HUS3_FA302_FF01_LM	AT%MX4202.1	:BOOL; 	(*	HUS3_FA302_FF01_LM	AS01	GVL.HUS3_FA302_FF01_LM	DIGITAL	0	0	0	0			Frånluftsfläkt ej i AUTO	p:B		*)	
	HUS3_FA302_GT51_LG	AT%MX4202.2	:BOOL; 	(*	HUS3_FA302_GT51_LG	AS01	GVL.HUS3_FA302_GT51_LG	DIGITAL	0	0	0	0			Givarfel frånluftsgivare	p:B		*)	
	HUS3_FA302_GT51_LH	AT%MX4202.3	:BOOL; 	(*	HUS3_FA302_GT51_LH	AS01	GVL.HUS3_FA302_GT51_LH	DIGITAL	0	0	0	0			Hög temperatur	p:B		*)	
																			
	HUS3_FA302_FF01_ACK	AT%MX4203.0	:BOOL; 	(*	HUS3_FA302_FF01_ACK	AS01	GVL.HUS3_FA302_FF01_ACK	DIGITAL	0	0	0	0			Larmkvittens frånluftsfläkt			*)
																			
																			
	HUS3_FA303_SO1_LM	AT%MX4204.0	:BOOL; 	(*	HUS3_FA303_SO1_LM	AS01	GVL.HUS3_FA303_SO1_LM	DIGITAL	0	0	0	0			Serviceomkopplare ej i läge AUTO	p:C		*)	
	HUS3_FA303_FF01_LM	AT%MX4204.1	:BOOL; 	(*	HUS3_FA303_FF01_LM	AS01	GVL.HUS3_FA303_FF01_LM	DIGITAL	0	0	0	0			Frånluftsfläkt ej i AUTO	p:B		*)	
	HUS3_FA303_GT51_LG	AT%MX4204.2	:BOOL; 	(*	HUS3_FA303_GT51_LG	AS01	GVL.HUS3_FA303_GT51_LG	DIGITAL	0	0	0	0			Givarfel frånluftsgivare	p:B		*)	
	HUS3_FA303_GT51_LH	AT%MX4204.3	:BOOL; 	(*	HUS3_FA303_GT51_LH	AS01	GVL.HUS3_FA303_GT51_LH	DIGITAL	0	0	0	0			Hög temperatur	p:B		*)	
																			
	HUS3_FA303_FF01_ACK	AT%MX4205.0	:BOOL; 	(*	HUS3_FA303_FF01_ACK	AS01	GVL.HUS3_FA303_FF01_ACK	DIGITAL	0	0	0	0			Larmkvittens frånluftsfläkt			*)
																			
																			
																			
																			




END_VAR

(* Global variable list: HUS3/FA301, FA302, FA303/HUS3_FA301_303_OVRIGT *)
VAR_GLOBAL



																						
	HUS3_FA301_SO1_IH	AT%MX4210.0	:BOOL;	(*	HUS3_FA301_SO1_IH	AS01	GVL.HUS3_FA301_SO1_IH	DIGITAL	0	0	0	0			Serviceomkopplare ej i AUTO			*)				
	HUS3_FA301_SO1_IA	AT%MX4210.1	:BOOL;	(*	HUS3_FA301_SO1_IA	AS01	GVL.HUS3_FA301_SO1_IA	DIGITAL	0	0	0	0			Serviceomkopplare i läge AUTO			*)				
	HUS3_FA301_SO1_IF	AT%MX4210.2	:BOOL;	(*	HUS3_FA301_SO1_IF	AS01	GVL.HUS3_FA301_SO1_IF	DIGITAL	0	0	0	0			Serviceomkopplare i läge 0			*)				
	HUS3_FA301_SO1_IT	AT%MX4210.3	:BOOL;	(*	HUS3_FA301_SO1_IT	AS01	GVL.HUS3_FA301_SO1_IT	DIGITAL	0	0	0	0			Serviceomkopplare i läge HAND TILL			*)				
																						
	HUS3_FA301_FF01_IT	AT%MX4210.5	:BOOL;	(*	HUS3_FA301_FF01_IT	AS01	GVL.HUS3_FA301_FF01_IT	DIGITAL	0	0	0	0			Frånluftsfläkt indikering TILL			*)				
																						
																						
	HUS3_FA302_SO1_IH	AT%MX4211.0	:BOOL;	(*	HUS3_FA302_SO1_IH	AS01	GVL.HUS3_FA302_SO1_IH	DIGITAL	0	0	0	0			Serviceomkopplare ej i AUTO			*)				
	HUS3_FA302_SO1_IA	AT%MX4211.1	:BOOL;	(*	HUS3_FA302_SO1_IA	AS01	GVL.HUS3_FA302_SO1_IA	DIGITAL	0	0	0	0			Serviceomkopplare i läge AUTO			*)				
	HUS3_FA302_SO1_IF	AT%MX4211.2	:BOOL;	(*	HUS3_FA302_SO1_IF	AS01	GVL.HUS3_FA302_SO1_IF	DIGITAL	0	0	0	0			Serviceomkopplare i läge 0			*)				
	HUS3_FA302_SO1_IT	AT%MX4211.3	:BOOL;	(*	HUS3_FA302_SO1_IT	AS01	GVL.HUS3_FA302_SO1_IT	DIGITAL	0	0	0	0			Serviceomkopplare i läge HAND TILL			*)				
																						
	HUS3_FA302_FF01_IT	AT%MX4211.5	:BOOL;	(*	HUS3_FA302_FF01_IT	AS01	GVL.HUS3_FA302_FF01_IT	DIGITAL	0	0	0	0			Frånluftsfläkt indikering TILL			*)				
																						
																						
	HUS3_FA303_SO1_IH	AT%MX4212.0	:BOOL;	(*	HUS3_FA303_SO1_IH	AS01	GVL.HUS3_FA303_SO1_IH	DIGITAL	0	0	0	0			Serviceomkopplare ej i AUTO			*)				
	HUS3_FA303_SO1_IA	AT%MX4212.1	:BOOL;	(*	HUS3_FA303_SO1_IA	AS01	GVL.HUS3_FA303_SO1_IA	DIGITAL	0	0	0	0			Serviceomkopplare i läge AUTO			*)				
	HUS3_FA303_SO1_IF	AT%MX4212.2	:BOOL;	(*	HUS3_FA303_SO1_IF	AS01	GVL.HUS3_FA303_SO1_IF	DIGITAL	0	0	0	0			Serviceomkopplare i läge 0			*)				
	HUS3_FA303_SO1_IT	AT%MX4212.3	:BOOL;	(*	HUS3_FA303_SO1_IT	AS01	GVL.HUS3_FA303_SO1_IT	DIGITAL	0	0	0	0			Serviceomkopplare i läge HAND TILL			*)				
																						
	HUS3_FA303_FF01_IT	AT%MX4212.5	:BOOL;	(*	HUS3_FA303_FF01_IT	AS01	GVL.HUS3_FA303_FF01_IT	DIGITAL	0	0	0	0			Frånluftsfläkt indikering TILL			*)				
																						
																						
																						



END_VAR

(* Global variable list: HUS3/VS40/HUS3_VS40_INST *)
VAR_GLOBAL PERSISTENT


																					
				(*	Name	Device	Address	Data type	Rawmin	Rawmax	Engmin	Engmax	Unit	Format	Description	Alarmoptions	Trendoptions	*)			
																					
	HUS3_VS40_GT11_UX1	AT%MB3692	:REAL;	(*	HUS3_VS40_GT11_UX1	AS01	GVL.HUS3_VS40_GT11_UX1	REAL	-50	150	-50	150	°C	0.0	Utetemp. kompenserad kurva Brytpunkt X1			*)			
	HUS3_VS40_GT11_UX2	AT%MB3696	:REAL;	(*	HUS3_VS40_GT11_UX2	AS01	GVL.HUS3_VS40_GT11_UX2	REAL	-50	150	-50	150	°C	0.0	Utetemp. kompenserad kurva Brytpunkt X2			*)			
	HUS3_VS40_GT11_UX3	AT%MB3700	:REAL;	(*	HUS3_VS40_GT11_UX3	AS01	GVL.HUS3_VS40_GT11_UX3	REAL	-50	150	-50	150	°C	0.0	Utetemp. kompenserad kurva Brytpunkt X3			*)			
	HUS3_VS40_GT11_UX4	AT%MB3704	:REAL;	(*	HUS3_VS40_GT11_UX4	AS01	GVL.HUS3_VS40_GT11_UX4	REAL	-50	150	-50	150	°C	0.0	Utetemp. kompenserad kurva Brytpunkt X4			*)			
	HUS3_VS40_GT11_UX5	AT%MB3708	:REAL;	(*	HUS3_VS40_GT11_UX5	AS01	GVL.HUS3_VS40_GT11_UX5	REAL	-50	150	-50	150	°C	0.0	Utetemp. kompenserad kurva Brytpunkt X5			*)			
	HUS3_VS40_GT11_UY1	AT%MB3712	:REAL;	(*	HUS3_VS40_GT11_UY1	AS01	GVL.HUS3_VS40_GT11_UY1	REAL	0	150	0	150	°C	0.0	Utetemp. kompenserad kurva Brytpunkt Y1			*)			
	HUS3_VS40_GT11_UY2	AT%MB3716	:REAL;	(*	HUS3_VS40_GT11_UY2	AS01	GVL.HUS3_VS40_GT11_UY2	REAL	0	150	0	150	°C	0.0	Utetemp. kompenserad kurva Brytpunkt Y2			*)			
	HUS3_VS40_GT11_UY3	AT%MB3720	:REAL;	(*	HUS3_VS40_GT11_UY3	AS01	GVL.HUS3_VS40_GT11_UY3	REAL	0	150	0	150	°C	0.0	Utetemp. kompenserad kurva Brytpunkt Y3			*)			
	HUS3_VS40_GT11_UY4	AT%MB3724	:REAL;	(*	HUS3_VS40_GT11_UY4	AS01	GVL.HUS3_VS40_GT11_UY4	REAL	0	150	0	150	°C	0.0	Utetemp. kompenserad kurva Brytpunkt Y4			*)			
	HUS3_VS40_GT11_UY5	AT%MB3728	:REAL;	(*	HUS3_VS40_GT11_UY5	AS01	GVL.HUS3_VS40_GT11_UY5	REAL	0	150	0	150	°C	0.0	Utetemp. kompenserad kurva Brytpunkt Y5			*)			
	HUS3_VS40_GT11_UMIN	AT%MB3732	:REAL;	(*	HUS3_VS40_GT11_UMIN	AS01	GVL.HUS3_VS40_GT11_UMIN	REAL	0	150	0	150	°C	0.0	Utetemp. kompenserad kurva Min-begränsning			*)			
	HUS3_VS40_GT11_UMAX	AT%MB3736	:REAL;	(*	HUS3_VS40_GT11_UMAX	AS01	GVL.HUS3_VS40_GT11_UMAX	REAL	0	150	0	150	°C	0.0	Utetemp. kompenserad kurva Max-begränsning			*)			
																					
	HUS3_VS40_GT11_CP	AT%MB3740	:REAL;	(*	HUS3_VS40_GT11_CPV	AS01	GVL.HUS3_VS40_GT11_CP	REAL	0	10	0	10		0.0	P-parameter			*)			
	HUS3_VS40_GT11_CI	AT%MB3744	:REAL;	(*	HUS3_VS40_GT11_CIV	AS01	GVL.HUS3_VS40_GT11_CI	REAL	0	900	0	900	Sek		I-Tid 			*)			
	HUS3_VS40_GT11_CD	AT%MB3748	:REAL;	(*	HUS3_VS40_GT11_CDV	AS01	GVL.HUS3_VS40_GT11_CD	REAL	0	900	0	900	Sek		D-tid 			*)			
	HUS3_VS40_GT11_CS	AT%MB3752	:REAL;	(*	HUS3_VS40_GT11_CSV	AS01	GVL.HUS3_VS40_GT11_CS	REAL	0	900	0	900	Sek		Samplingstid			*)			
	HUS3_VS40_GT11_CZ	AT%MB3756	:REAL;	(*	HUS3_VS40_GT11_CZV	AS01	GVL.HUS3_VS40_GT11_CZ	REAL	-10	10	-10	10	°C	0.0	Dödband regulator			*)			
																					
	HUS3_VS40_SO1_MAN	AT%MB3760	:INT;	(*	HUS3_VS40_SO1_MAN	AS01	GVL.HUS3_VS40_SO1_MAN	INT	0	2	0	2			Manuell styrning system VS40. 0=Auto, 1=Manuell från, 2=Manuell till			*)			
	HUS3_VS40_PV01_MAN	AT%MB3762	:INT;	(*	HUS3_VS40_PV01_MAN	AS01	GVL.HUS3_VS40_PV01_MAN	INT	0	2	0	2			Manuell styrning crikulationspump 0=Auto,1=Från,2=Till			*)			
	HUS3_VS40_SV21_MAN1	AT%MB3764	:INT;	(*	HUS3_VS40_SV21_MAN	AS01	GVL.HUS3_VS40_SV21_MAN	INT	0	1	0	1			Manuell styrning ventilställdon 0=Auto,1=Hand			*)			
	HUS3_VS40_SV21_RMAN	AT%MB3768	:REAL;	(*	HUS3_VS40_SV21_RMAN	AS01	GVL.HUS3_VS40_SV21_RMAN	REAL	0	100	0	100	%		Manuell styrsignal ventilställdon			*)			
																					
	HUS3_VS40_SO1_FLM	AT%MB3772	:INT;	(*	HUS3_VS40_SO1_FLM	AS01	GVL.HUS3_VS40_SO1_FLM	INT	0	3600	0	3600	Min		Larmfördröjning serviceomkopplare ej i läge AUTO			*)			
	HUS3_VS40_PV01_FLM	AT%MB3774	:INT;	(*	HUS3_VS40_PV01_FLM	AS01	GVL.HUS3_VS40_PV01_FLM	INT	0	3600	0	3600	Min		Larmfördröjning cirkulationspump ej i AUTO			*)			
	HUS3_VS40_SV21_FLM	AT%MB3776	:INT;	(*	HUS3_VS40_SV21_FLM	AS01	GVL.HUS3_VS40_SV21_FLM	INT	0	3600	0	3600	Min		Larmfördröjning ventilställdon ej i AUTO			*)			
	HUS3_VS40_PV01_FLD	AT%MB3778	:INT;	(*	HUS3_VS40_PV01_FLD	AS01	GVL.HUS3_VS40_PV01_FLD	INT	0	120	0	120	Sek		Larmfördröjning driftfel cirkulationspump			*)			
																					
	HUS3_VS40_GT11_GAVH	AT%MB3784	:REAL;	(*	HUS3_VS40_GT11_GAVH	AS01	GVL.HUS3_VS40_GT11_GAVH	REAL	-20	20	-20	20	°C	0.0	Gränsavvikelse hög framledningstemperatur			*)			
	HUS3_VS40_GT11_GAVL	AT%MB3788	:REAL;	(*	HUS3_VS40_GT11_GAVL	AS01	GVL.HUS3_VS40_GT11_GAVL	REAL	-20	20	-20	20	°C	0.0	Gränsavvikelse låg framledningstemperatur			*)			
	HUS3_VS40_GT11_FLAH	AT%MB3792	:INT;	(*	HUS3_VS40_GT11_FLAH	AS01	GVL.HUS3_VS40_GT11_FLAH	INT	0	3600	0	3600	Min		Larmfördröjning hög framledningstemperatur			*)			
	HUS3_VS40_GT11_FLAL	AT%MB3794	:INT;	(*	HUS3_VS40_GT11_FLAL	AS01	GVL.HUS3_VS40_GT11_FLAL	INT	0	3600	0	3600	Min		Lamfördröjning låg framledningstemperatur			*)			
																					
																					
																					
																					
																					
																					
																					
																					
																					
	HUS3_VS40_GT11_KRV	AT%MB3796	:REAL;	(*	HUS3_VS40_GT11_KRV	AS01	GVL.HUS3_VS40_GT11_KRV	REAL	-10	10	-10	10	°C	0.0	Kalibreringsvärde framledningsgivare			*)			
	HUS3_VS40_GT41_KRV	AT%MB3800	:REAL;	(*	HUS3_VS40_GT41_KRV	AS01	GVL.HUS3_VS40_GT41_KRV	REAL	-10	10	-10	10	°C	0.0	Kalibreringsvärde returgivare			*)			
																					
																					
																					
	HUS3_VS40_GT11_X1	AT%MB3804	:REAL;	(*	HUS3_VS40_GT11_X1	AS01	GVL.HUS3_VS40_GT11_X1	REAL	-50	150	-50	150	°C	0.0	Effektbegränsning kurva Brytpunkt X1			*)			
	HUS3_VS40_GT11_X2	AT%MB3808	:REAL;	(*	HUS3_VS40_GT11_X2	AS01	GVL.HUS3_VS40_GT11_X2	REAL	-50	150	-50	150	°C	0.0	Effektbegränsning kurva Brytpunkt X2			*)			
	HUS3_VS40_GT11_X3	AT%MB3812	:REAL;	(*	HUS3_VS40_GT11_X3	AS01	GVL.HUS3_VS40_GT11_X3	REAL	-50	150	-50	150	°C	0.0	Effektbegränsning kurva Brytpunkt X3			*)			
	HUS3_VS40_GT11_X4	AT%MB3816	:REAL;	(*	HUS3_VS40_GT11_X4	AS01	GVL.HUS3_VS40_GT11_X4	REAL	-50	150	-50	150	°C	0.0	Effektbegränsning kurva Brytpunkt X4			*)			
	HUS3_VS40_GT11_X5	AT%MB3820	:REAL;	(*	HUS3_VS40_GT11_X5	AS01	GVL.HUS3_VS40_GT11_X5	REAL	-50	150	-50	150	°C	0.0	Effektbegränsning kurva Brytpunkt X5			*)			
	HUS3_VS40_GT11_Y1	AT%MB3824	:REAL;	(*	HUS3_VS40_GT11_Y1	AS01	GVL.HUS3_VS40_GT11_Y1	REAL	0	150	0	150	°C	0.0	Effektbegränsning kurva Brytpunkt Y1			*)			
	HUS3_VS40_GT11_Y2	AT%MB3828	:REAL;	(*	HUS3_VS40_GT11_Y2	AS01	GVL.HUS3_VS40_GT11_Y2	REAL	0	150	0	150	°C	0.0	Effektbegränsning kurva Brytpunkt Y2			*)			
	HUS3_VS40_GT11_Y3	AT%MB3832	:REAL;	(*	HUS3_VS40_GT11_Y3	AS01	GVL.HUS3_VS40_GT11_Y3	REAL	0	150	0	150	°C	0.0	Effektbegränsning kurva Brytpunkt Y3			*)			
	HUS3_VS40_GT11_Y4	AT%MB3836	:REAL;	(*	HUS3_VS40_GT11_Y4	AS01	GVL.HUS3_VS40_GT11_Y4	REAL	0	150	0	150	°C	0.0	Effektbegränsning kurva Brytpunkt Y4			*)			
	HUS3_VS40_GT11_Y5	AT%MB3840	:REAL;	(*	HUS3_VS40_GT11_Y5	AS01	GVL.HUS3_VS40_GT11_Y5	REAL	0	150	0	150	°C	0.0	Effektbegränsning kurva Brytpunkt Y5			*)			
	HUS3_VS40_GT11_MIN	AT%MB3844	:REAL;	(*	HUS3_VS40_GT11_MIN	AS01	GVL.HUS3_VS40_GT11_MIN	REAL	0	150	0	150	°C	0.0	Effektbegränsning kurva Min-begränsning			*)			
	HUS3_VS40_GT11_MAX	AT%MB3848	:REAL;	(*	HUS3_VS40_GT11_MAX	AS01	GVL.HUS3_VS40_GT11_MAX	REAL	0	150	0	150	°C	0.0	Effektbegränsning kurva Max-begränsning			*)			
																					
																					
																					
																					
																					
																					
																					
																					
																					



END_VAR
																
																

(* Global variable list: HUS3/VS40/HUS3_VS40_LARM *)
VAR_GLOBAL




																									
																									
	HUS3_VS40_SO1_LM	AT%MX3854.0	:BOOL; 	(*	HUS3_VS40_SO1_LM	AS01	GVL.HUS3_VS40_SO1_LM	DIGITAL	0	0	0	0			Serviceomkopplare ej i läge AUTO	p:C		*)							
	HUS3_VS40_PV01_LM	AT%MX3854.1	:BOOL; 	(*	HUS3_VS40_PV01_LM	AS01	GVL.HUS3_VS40_PV01_LM	DIGITAL	0	0	0	0			Cirkulationspump ej i AUTO	p:B		*)							
	HUS3_VS40_SV21_LM	AT%MX3854.2	:BOOL; 	(*	HUS3_VS40_SV21_LM	AS01	GVL.HUS3_VS40_SV21_LM	DIGITAL	0	0	0	0			Ventilställdon ej i AUTO	p:B		*)							
	HUS3_VS40_PV01_LD	AT%MX3854.3	:BOOL; 	(*	HUS3_VS40_PV01_LD	AS01	GVL.HUS3_VS40_PV01_LD	DIGITAL	0	0	0	0			Driftfel cirkulationspump	p:B		*)							
	HUS3_VS40_GT11_LG	AT%MX3854.4	:BOOL; 	(*	HUS3_VS40_GT11_LG	AS01	GVL.HUS3_VS40_GT11_LG	DIGITAL	0	0	0	0			Givarfel framledningsgivare	p:B		*)							
	HUS3_VS40_GT41_LG	AT%MX3854.5	:BOOL; 	(*	HUS3_VS40_GT41_LG	AS01	GVL.HUS3_VS40_GT41_LG	DIGITAL	0	0	0	0			Givarfel returgivare	p:B		*)							
	HUS3_VS40_GT11_LAH	AT%MX3854.6	:BOOL; 	(*	HUS3_VS40_GT11_LAH	AS01	GVL.HUS3_VS40_GT11_LAH	DIGITAL	0	0	0	0			Larmavvikelse hög framledningstemp	p:B		*)							
	HUS3_VS40_GT11_LAL	AT%MX3854.7	:BOOL; 	(*	HUS3_VS40_GT11_LAL	AS01	GVL.HUS3_VS40_GT11_LAL	DIGITAL	0	0	0	0			Larmavvikelse låg framledningstemp	p:B		*)							
																									
																									
																									
																									
																									
																									
																									
																									
																									
																									
																									
	HUS3_VS40_PV01_ACK	AT%MX3858.0	:BOOL; 	(*	HUS3_VS40_PV01_ACK	AS01	GVL.HUS3_VS40_PV01_ACK	DIGITAL	0	0	0	0			Larmkvittens pump			*)							
																									
																									
																									
																									
																									
																									
																									




END_VAR

(* Global variable list: HUS3/VS40/HUS3_VS40_OVRIGT *)
VAR_GLOBAL




																						
	HUS3_VS40_SO1_IH	AT%MX3860.0	:BOOL;	(*	HUS3_VS40_SO1_IH	AS01	GVL.HUS3_VS40_SO1_IH	DIGITAL	0	0	0	0			Serviceomkopplare ej i AUTO			*)				
	HUS3_VS40_SO1_IA	AT%MX3860.1	:BOOL;	(*	HUS3_VS40_SO1_IA	AS01	GVL.HUS3_VS40_SO1_IA	DIGITAL	0	0	0	0			Serviceomkopplare i läge AUTO			*)				
	HUS3_VS40_SO1_IF	AT%MX3860.2	:BOOL;	(*	HUS3_VS40_SO1_IF	AS01	GVL.HUS3_VS40_SO1_IF	DIGITAL	0	0	0	0			Serviceomkopplare i läge 0			*)				
	HUS3_VS40_SO1_IT	AT%MX3860.3	:BOOL;	(*	HUS3_VS40_SO1_IT	AS01	GVL.HUS3_VS40_SO1_IT	DIGITAL	0	0	0	0			Serviceomkopplare i läge HAND TILL			*)				
																						
																						
																						
																						
																						
																						
																						
																						
																						
																						
																						
																						
	HUS3_VS40_GT11_BB	AT%MB3864	:REAL;	(*	HUS3_VS40_GT11_BB	AS01	GVL.HUS3_VS40_GT11_BB	REAL	0	150	0	150	°C	0.0	Beräknat börvärde framledningstemperatur			*)				
	HUS3_VS40_GT11_BB1	AT%MB3868	:REAL;	(*	HUS3_VS40_GT11_BB1	AS01	GVL.HUS3_VS40_GT11_BB1	REAL	0	150	0	150	°C	0.0	Beräknad förskjutning framledningstemperatur			*)				
																						
																						
																						
																						
																						
																						

																						

																					

END_VAR

(* Global variable list: LB01-LB06/LB01_LB06_INST *)
VAR_GLOBAL PERSISTENT

																			
					(*	Name	Device	Address	Data type	Rawmin	Rawmax	Engmin	Engmax	Unit	Format	Description	Alarmoptions	Trendoptions	*)
																			
																			
		HUS1_LB01_GP11_BV	AT%MB5000	:REAL;	(*	HUS1_LB01_GP11_BV	AS01	GVL.HUS1_LB01_GP11_BV	REAL	0	1000	0	1000	Pa		Tryckbörvärde tilluft högfart			*)
		HUS1_LB01_GP12_BV	AT%MB5004	:REAL;	(*	HUS1_LB01_GP12_BV	AS01	GVL.HUS1_LB01_GP12_BV	REAL	0	1000	0	1000	Pa		Tryckbörvärde frånluft högfart			*)
		HUS1_LB01_GT11_BV	AT%MB5008	:REAL;	(*	HUS1_LB01_GT11_BV	AS01	GVL.HUS1_LB01_GT11_BV	REAL	0	50	0	50	°C	0.0	Temperaturbörvärde tilluft			*)
		HUS1_LB02_GP11_BV	AT%MB5012	:REAL;	(*	HUS1_LB02_GP11_BV	AS01	GVL.HUS1_LB02_GP11_BV	REAL	0	1000	0	1000	Pa		Tryckbörvärde tilluft högfart			*)
		HUS1_LB02_GP12_BV	AT%MB5016	:REAL;	(*	HUS1_LB02_GP12_BV	AS01	GVL.HUS1_LB02_GP12_BV	REAL	0	1000	0	1000	Pa		Tryckbörvärde frånluft högfart			*)
		HUS1_LB02_GT11_BV	AT%MB5020	:REAL;	(*	HUS1_LB02_GT11_BV	AS01	GVL.HUS1_LB02_GT11_BV	REAL	0	50	0	50	°C	0.0	Temperaturbörvärde tilluft			*)
		HUS2_LB03_GP11_BV	AT%MB5024	:REAL;	(*	HUS2_LB03_GP11_BV	AS01	GVL.HUS2_LB03_GP11_BV	REAL	0	1000	0	1000	Pa		Tryckbörvärde tilluft högfart			*)
		HUS2_LB03_GP12_BV	AT%MB5028	:REAL;	(*	HUS2_LB03_GP12_BV	AS01	GVL.HUS2_LB03_GP12_BV	REAL	0	1000	0	1000	Pa		Tryckbörvärde frånluft högfart			*)
		HUS2_LB03_GT11_BV	AT%MB5032	:REAL;	(*	HUS2_LB03_GT11_BV	AS01	GVL.HUS2_LB03_GT11_BV	REAL	0	50	0	50	°C	0.0	Temperaturbörvärde tilluft			*)
		HUS3_LB04_GP11_BV	AT%MB5036	:REAL;	(*	HUS3_LB04_GP11_BV	AS01	GVL.HUS3_LB04_GP11_BV	REAL	0	1000	0	1000	Pa		Tryckbörvärde tilluft högfart			*)
		HUS3_LB04_GP12_BV	AT%MB5040	:REAL;	(*	HUS3_LB04_GP12_BV	AS01	GVL.HUS3_LB04_GP12_BV	REAL	0	1000	0	1000	Pa		Tryckbörvärde frånluft högfart			*)
		HUS3_LB04_GT11_BV	AT%MB5044	:REAL;	(*	HUS3_LB04_GT11_BV	AS01	GVL.HUS3_LB04_GT11_BV	REAL	0	50	0	50	°C	0.0	Temperaturbörvärde tilluft			*)
		HUS3_LB05_GP11_BV	AT%MB5048	:REAL;	(*	HUS3_LB05_GP11_BV	AS01	GVL.HUS3_LB05_GP11_BV	REAL	0	1000	0	1000	Pa		Tryckbörvärde tilluft högfart			*)
		HUS3_LB05_GP12_BV	AT%MB5052	:REAL;	(*	HUS3_LB05_GP12_BV	AS01	GVL.HUS3_LB05_GP12_BV	REAL	0	1000	0	1000	Pa		Tryckbörvärde frånluft högfart			*)
		HUS3_LB05_GT11_BV	AT%MB5056	:REAL;	(*	HUS3_LB05_GT11_BV	AS01	GVL.HUS3_LB05_GT11_BV	REAL	0	50	0	50	°C	0.0	Temperaturbörvärde tilluft			*)
		HUS1_LB06_GP11_BVL	AT%MB5060	:REAL;	(*	HUS1_LB06_GP11_BVL	AS01	GVL.HUS1_LB06_GP11_BVL	REAL	0	1000	0	1000	Pa		Tryckbörvärde tilluft lågfart			*)
		HUS1_LB06_GP12_BVL	AT%MB5064	:REAL;	(*	HUS1_LB06_GP12_BVL	AS01	GVL.HUS1_LB06_GP12_BVL	REAL	0	1000	0	1000	Pa		Tryckbörvärde frånluft lågfart			*)
		HUS1_LB06_GP11_BVH	AT%MB5068	:REAL;	(*	HUS1_LB06_GP11_BVH	AS01	GVL.HUS1_LB06_GP11_BVGVL.H	REAL	0	1000	0	1000	Pa		Tryckbörvärde tilluft lågfart			*)
		HUS1_LB06_GP12_BVH	AT%MB5072	:REAL;	(*	HUS1_LB06_GP12_BVH	AS01	GVL.HUS1_LB06_GP12_BVGVL.H	REAL	0	1000	0	1000	Pa		Tryckbörvärde frånluft lågfart			*)
		HUS1_LB06_GT41_BV	AT%MB5076	:REAL;	(*	HUS1_LB06_GT41_BV	AS01	GVL.HUS1_LB06_GT41_BV	REAL	0	50	0	50	°C	0.0	Temperaturbörvärde frånluft			*)
		HUS1_LB06_GT11_BVMIN	AT%MB5080	:REAL;	(*	HUS1_LB06_GT11_BVMIN	AS01	GVL.HUS1_LB06_GT11_BVMIN	REAL	0	50	0	50	°C	0.0	Temperaturbörvärde tilluft MIN			*)
		HUS1_LB06_GT11_BVMAX	AT%MB5084	:REAL;	(*	HUS1_LB06_GT11_BVMAX	AS01	GVL.HUS1_LB06_GT11_BVMAX	REAL	0	50	0	50	°C	0.0	Temperaturbörvärde tilluft MAX			*)
																			
																			
																			
		HUS1_LB01_LC_FL	AT%MB5088	:INT;	(*	HUS1_LB01_LC_FL	AS01	GVL.HUS1_LB01_LC_FL	INT	0	3600	0	3600	min		Larmfördröjning kommunikationsfel			*)
		HUS1_LB02_LC_FL	AT%MB5090	:INT;	(*	HUS1_LB02_LC_FL	AS01	GVL.HUS1_LB02_LC_FL	INT	0	3600	0	3600	min		Larmfördröjning kommunikationsfel			*)
		HUS2_LB03_LC_FL	AT%MB5092	:INT;	(*	HUS2_LB03_LC_FL	AS01	GVL.HUS2_LB03_LC_FL	INT	0	3600	0	3600	min		Larmfördröjning kommunikationsfel			*)
		HUS3_LB04_LC_FL	AT%MB5094	:INT;	(*	HUS3_LB04_LC_FL	AS01	GVL.HUS3_LB04_LC_FL	INT	0	3600	0	3600	min		Larmfördröjning kommunikationsfel			*)
		HUS3_LB05_LC_FL	AT%MB5096	:INT;	(*	HUS3_LB05_LC_FL	AS01	GVL.HUS3_LB05_LC_FL	INT	0	3600	0	3600	min		Larmfördröjning kommunikationsfel			*)
		HUS1_LB06_LC_FL	AT%MB5098	:INT;	(*	HUS1_LB06_LC_FL	AS01	GVL.HUS1_LB06_LC_FL	INT	0	3600	0	3600	min		Larmfördröjning kommunikationsfel			*)
																			
																			
																			



END_VAR

(* Global variable list: LB01-LB06/LB01_LB06_OVRIGT *)
VAR_GLOBAL


	(*LARM*)																			
																				
		HUS1_LB01_LC	AT%MX5120.0	:BOOL; 	(*	HUS1_LB01_LC	AS01	GVL.HUS1_LB01_LC	DIGITAL	0	0	0	0			Kommunikationsfel	p:B		*)	
		HUS1_LB01_L1	AT%MX5120.1	:BOOL; 	(*	HUS1_LB01_L1	AS01	GVL.HUS1_LB01_L1	DIGITAL	0	0	0	0			Summalarm A	p:A		*)	
		HUS1_LB01_L2	AT%MX5120.2	:BOOL; 	(*	HUS1_LB01_L2	AS01	GVL.HUS1_LB01_L2	DIGITAL	0	0	0	0			Summalarm B	p:B		*)	
		HUS1_LB02_LC	AT%MX5120.3	:BOOL; 	(*	HUS1_LB02_LC	AS01	GVL.HUS1_LB02_LC	DIGITAL	0	0	0	0			Kommunikationsfel	p:B		*)	
		HUS1_LB02_L1	AT%MX5120.4	:BOOL; 	(*	HUS1_LB02_L1	AS01	GVL.HUS1_LB02_L1	DIGITAL	0	0	0	0			Summalarm A	p:A		*)	
		HUS1_LB02_L2	AT%MX5120.5	:BOOL; 	(*	HUS1_LB02_L2	AS01	GVL.HUS1_LB02_L2	DIGITAL	0	0	0	0			Summalarm B	p:B		*)	
		HUS2_LB03_LC	AT%MX5120.6	:BOOL; 	(*	HUS2_LB03_LC	AS01	GVL.HUS2_LB03_LC	DIGITAL	0	0	0	0			Kommunikationsfel	p:B		*)	
		HUS2_LB03_L1	AT%MX5120.7	:BOOL; 	(*	HUS2_LB03_L1	AS01	GVL.HUS2_LB03_L1	DIGITAL	0	0	0	0			Summalarm A	p:A		*)	
		HUS2_LB03_L2	AT%MX5121.0	:BOOL; 	(*	HUS2_LB03_L2	AS01	GVL.HUS2_LB03_L2	DIGITAL	0	0	0	0			Summalarm B	p:B		*)	
		HUS3_LB04_LC	AT%MX5121.1	:BOOL; 	(*	HUS3_LB04_LC	AS01	GVL.HUS3_LB04_LC	DIGITAL	0	0	0	0			Kommunikationsfel	p:B		*)	
		HUS3_LB04_L1	AT%MX5121.2	:BOOL; 	(*	HUS3_LB04_L1	AS01	GVL.HUS3_LB04_L1	DIGITAL	0	0	0	0			Summalarm A	p:A		*)	
		HUS3_LB04_L2	AT%MX5121.3	:BOOL; 	(*	HUS3_LB04_L2	AS01	GVL.HUS3_LB04_L2	DIGITAL	0	0	0	0			Summalarm B	p:B		*)	
		HUS3_LB05_LC	AT%MX5121.4	:BOOL; 	(*	HUS3_LB05_LC	AS01	GVL.HUS3_LB05_LC	DIGITAL	0	0	0	0			Kommunikationsfel	p:B		*)	
		HUS3_LB05_L1	AT%MX5121.5	:BOOL; 	(*	HUS3_LB05_L1	AS01	GVL.HUS3_LB05_L1	DIGITAL	0	0	0	0			Summalarm A	p:A		*)	
		HUS3_LB05_L2	AT%MX5121.6	:BOOL; 	(*	HUS3_LB05_L2	AS01	GVL.HUS3_LB05_L2	DIGITAL	0	0	0	0			Summalarm B	p:B		*)	
		HUS1_LB06_LC	AT%MX5121.7	:BOOL; 	(*	HUS1_LB06_LC	AS01	GVL.HUS1_LB06_LC	DIGITAL	0	0	0	0			Kommunikationsfel	p:B		*)	
		HUS1_LB06_L1	AT%MX5122.0	:BOOL; 	(*	HUS1_LB06_L1	AS01	GVL.HUS1_LB06_L1	DIGITAL	0	0	0	0			Summalarm A	p:A		*)	
		HUS1_LB06_L2	AT%MX5122.1	:BOOL; 	(*	HUS1_LB06_L2	AS01	GVL.HUS1_LB06_L2	DIGITAL	0	0	0	0			Summalarm B	p:B		*)	
																				
																				

	(*ÖVRIGT, INDIKERINGAR, MÄTVÄRDEN*)																						
																							
		HUS1_LB01_PV01_IT	AT%MX5123.0	:BOOL; 	(*	HUS1_LB01_PV01_IT	AS01	GVL.HUS1_LB01_PV01_IT	DIGITAL	0	0	0	0			Crikulationspump indikering TILL			*)				
		HUS1_LB02_PV01_IT	AT%MX5123.1	:BOOL; 	(*	HUS1_LB02_PV01_IT	AS01	GVL.HUS1_LB02_PV01_IT	DIGITAL	0	0	0	0			Crikulationspump indikering TILL			*)				
		HUS2_LB03_PV01_IT	AT%MX5123.2	:BOOL; 	(*	HUS2_LB03_PV01_IT	AS01	GVL.HUS2_LB03_PV01_IT	DIGITAL	0	0	0	0			Crikulationspump indikering TILL			*)				
		HUS3_LB04_PV01_IT	AT%MX5123.3	:BOOL; 	(*	HUS3_LB04_PV01_IT	AS01	GVL.HUS3_LB04_PV01_IT	DIGITAL	0	0	0	0			Crikulationspump indikering TILL			*)				
		HUS3_LB05_PV01_IT	AT%MX5123.4	:BOOL; 	(*	HUS3_LB05_PV01_IT	AS01	GVL.HUS3_LB05_PV01_IT	DIGITAL	0	0	0	0			Crikulationspump indikering TILL			*)				
		HUS1_LB06_PV01_IT	AT%MX5123.5	:BOOL; 	(*	HUS1_LB06_PV01_IT	AS01	GVL.HUS1_LB06_PV01_IT	DIGITAL	0	0	0	0			Crikulationspump indikering TILL			*)				

		HUS1_LB01_DRIFTLAGE	AT%MB5130	:INT;	(*	HUS1_LB01_DRIFTLAGE	AS01	GVL.HUS1_LB01_DRIFTLAGE	REAL	0	40	0	40			Aktuellt driftläge			*)
		HUS1_LB02_DRIFTLAGE	AT%MB5132	:INT;	(*	HUS1_LB02_DRIFTLAGE	AS01	GVL.HUS1_LB02_DRIFTLAGE	REAL	0	40	0	40			Aktuellt driftläge			*)	
		HUS2_LB03_DRIFTLAGE	AT%MB5134	:INT;	(*	HUS2_LB03_DRIFTLAGE	AS01	GVL.HUS2_LB03_DRIFTLAGE	REAL	0	40	0	40			Aktuellt driftläge			*)	
		HUS3_LB04_DRIFTLAGE	AT%MB5136	:INT;	(*	HUS3_LB04_DRIFTLAGE	AS01	GVL.HUS3_LB04_DRIFTLAGE	REAL	0	40	0	40			Aktuellt driftläge			*)	
		HUS3_LB05_DRIFTLAGE	AT%MB5138	:INT;	(*	HUS3_LB05_DRIFTLAGE	AS01	GVL.HUS3_LB05_DRIFTLAGE	REAL	0	40	0	40			Aktuellt driftläge			*)	
		HUS1_LB06_DRIFTLAGE	AT%MB5140	:INT;	(*	HUS1_LB06_DRIFTLAGE	AS01	GVL.HUS1_LB06_DRIFTLAGE	REAL	0	40	0	40			Aktuellt driftläge			*)	
																				
		HUS1_LB01_GF41_MV	AT%MB5152	:REAL;	(*	HUS1_LB01_GF41_MV	AS01	GVL.HUS1_LB01_GF41_MV	REAL	0	4000	0	4000	l/s	0.0	Mätvärde flöde tilluft			*)	
		HUS1_LB01_GF42_MV	AT%MB5156	:REAL;	(*	HUS1_LB01_GF42_MV	AS01	GVL.HUS1_LB01_GF42_MV	REAL	0	4000	0	4000	l/s	0.0	Mätvärde flöde frånluft			*)	
		HUS1_LB01_GP11_MV	AT%MB5160	:REAL;	(*	HUS1_LB01_GP11_MV	AS01	GVL.HUS1_LB01_GP11_MV	REAL	0	1000	0	1000	Pa		Mätvärde tryck tilluft			*)	
		HUS1_LB01_GP12_MV	AT%MB5164	:REAL;	(*	HUS1_LB01_GP12_MV	AS01	GVL.HUS1_LB01_GP12_MV	REAL	0	1000	0	1000	Pa		Mätvärde tryck frånluft			*)	
		HUS1_LB01_GP61_MV	AT%MB5168	:REAL;	(*	HUS1_LB01_GP61_MV	AS01	GVL.HUS1_LB01_GP61_MV	REAL	0	1000	0	1000	Pa		Mätvärde tryckfall tilluftsfilter			*)	
		HUS1_LB01_GP61_GV	AT%MB5172	:REAL;	(*	HUS1_LB01_GP61_GV	AS01	GVL.HUS1_LB01_GP61_GV	REAL	0	1000	0	1000	Pa		Sluttryckfall tilluftsfilter			*)	
		HUS1_LB01_GP62_MV	AT%MB5176	:REAL;	(*	HUS1_LB01_GP62_MV	AS01	GVL.HUS1_LB01_GP62_MV	REAL	0	1000	0	1000	Pa		Mätvärde tryckfall frånluftsfilter			*)	
		HUS1_LB01_GP62_GV	AT%MB5180	:REAL;	(*	HUS1_LB01_GP62_GV	AS01	GVL.HUS1_LB01_GP62_GV	REAL	0	1000	0	1000	Pa		Sluttryckfall frånluftsfilter			*)	
		HUS1_LB01_TF01_R	AT%MB5184	:REAL;	(*	HUS1_LB01_TF01_R	AS01	GVL.HUS1_LB01_TF01_R	REAL	0	100	0	100	%	0.0	Styrsignal tilluftsfläkt			*)	
		HUS1_LB01_FF01_R	AT%MB5188	:REAL;	(*	HUS1_LB01_FF01_R	AS01	GVL.HUS1_LB01_FF01_R	REAL	0	100	0	100	%	0.0	Styrsignal frånluftsfläkt			*)	
		HUS1_LB01_SFP_MV	AT%MB5192	:REAL;	(*	HUS1_LB01_SFP_MV	AS01	GVL.HUS1_LB01_SFP_MV	REAL	0	100	0	100	kW/m3/s	0.0	SFP-värde			*)	
		HUS1_LB01_GT11_MV	AT%MB5196	:REAL;	(*	HUS1_LB01_GT11_MV	AS01	GVL.HUS1_LB01_GT11_MV	REAL	-50	100	-50	100	°C	0.0	Mätvärde temperatur tilluft			*)	
		HUS1_LB01_GT41_MV	AT%MB5200	:REAL;	(*	HUS1_LB01_GT41_MV	AS01	GVL.HUS1_LB01_GT41_MV	REAL	-50	100	-50	100	°C	0.0	Mätvärde temperatur frånluft			*)	
		HUS1_LB01_GT31_MV	AT%MB5204	:REAL;	(*	HUS1_LB01_GT31_MV	AS01	GVL.HUS1_LB01_GT31_MV	REAL	-50	100	-50	100	°C	0.0	Mätvärde temperatur uteluft			*)	
		HUS1_LB01_GT81_MV	AT%MB5208	:REAL;	(*	HUS1_LB01_GT81_MV	AS01	GVL.HUS1_LB01_GT81_MV	REAL	-50	100	-50	100	°C	0.0	Mätvärde temperatur frysvakt			*)	
		HUS1_LB01_VVX01_VVX	AT%MB5212	:REAL;	(*	HUS1_LB01_VVX01_VVX	AS01	GVL.HUS1_LB01_VVX01_VVX	REAL	0	100	0	100	%	0.0	Verkningsgrad VVX			*)	
		HUS1_LB01_SV21_R	AT%MB5216	:REAL;	(*	HUS1_LB01_SV21_R	AS01	GVL.HUS1_LB01_SV21_R	REAL	0	100	0	100	%	0.0	Styrsignal ventilställdon värme			*)	
		HUS1_LB02_GF41_MV	AT%MB5220	:REAL;	(*	HUS1_LB02_GF41_MV	AS01	GVL.HUS1_LB02_GF41_MV	REAL	0	4000	0	4000	l/s	0.0	Mätvärde flöde tilluft			*)	
		HUS1_LB02_GF42_MV	AT%MB5224	:REAL;	(*	HUS1_LB02_GF42_MV	AS01	GVL.HUS1_LB02_GF42_MV	REAL	0	4000	0	4000	l/s	0.0	Mätvärde flöde frånluft			*)	
		HUS1_LB02_GP11_MV	AT%MB5228	:REAL;	(*	HUS1_LB02_GP11_MV	AS01	GVL.HUS1_LB02_GP11_MV	REAL	0	1000	0	1000	Pa		Mätvärde tryck tilluft			*)	
		HUS1_LB02_GP12_MV	AT%MB5232	:REAL;	(*	HUS1_LB02_GP12_MV	AS01	GVL.HUS1_LB02_GP12_MV	REAL	0	1000	0	1000	Pa		Mätvärde tryck frånluft			*)	
		HUS1_LB02_GP61_MV	AT%MB5236	:REAL;	(*	HUS1_LB02_GP61_MV	AS01	GVL.HUS1_LB02_GP61_MV	REAL	0	1000	0	1000	Pa		Mätvärde tryckfall tilluftsfilter			*)	
		HUS1_LB02_GP61_GV	AT%MB5240	:REAL;	(*	HUS1_LB02_GP61_GV	AS01	GVL.HUS1_LB02_GP61_GV	REAL	0	1000	0	1000	Pa		Sluttryckfall tilluftsfilter			*)	
		HUS1_LB02_GP62_MV	AT%MB5244	:REAL;	(*	HUS1_LB02_GP62_MV	AS01	GVL.HUS1_LB02_GP62_MV	REAL	0	1000	0	1000	Pa		Mätvärde tryckfall frånluftsfilter			*)	
		HUS1_LB02_GP62_GV	AT%MB5248	:REAL;	(*	HUS1_LB02_GP62_GV	AS01	GVL.HUS1_LB02_GP62_GV	REAL	0	1000	0	1000	Pa		Sluttryckfall frånluftsfilter			*)	
		HUS1_LB02_TF01_R	AT%MB5252	:REAL;	(*	HUS1_LB02_TF01_R	AS01	GVL.HUS1_LB02_TF01_R	REAL	0	100	0	100	%	0.0	Styrsignal tilluftsfläkt			*)	
		HUS1_LB02_FF01_R	AT%MB5256	:REAL;	(*	HUS1_LB02_FF01_R	AS01	GVL.HUS1_LB02_FF01_R	REAL	0	100	0	100	%	0.0	Styrsignal frånluftsfläkt			*)	
		HUS1_LB02_SFP_MV	AT%MB5260	:REAL;	(*	HUS1_LB02_SFP_MV	AS01	GVL.HUS1_LB02_SFP_MV	REAL	0	100	0	100	kW/m3/s	0.0	SFP-värde			*)	
		HUS1_LB02_GT11_MV	AT%MB5264	:REAL;	(*	HUS1_LB02_GT11_MV	AS01	GVL.HUS1_LB02_GT11_MV	REAL	-50	100	-50	100	°C	0.0	Mätvärde temperatur tilluft			*)	
		HUS1_LB02_GT41_MV	AT%MB5268	:REAL;	(*	HUS1_LB02_GT41_MV	AS01	GVL.HUS1_LB02_GT41_MV	REAL	-50	100	-50	100	°C	0.0	Mätvärde temperatur frånluft			*)	
		HUS1_LB02_GT31_MV	AT%MB5272	:REAL;	(*	HUS1_LB02_GT31_MV	AS01	GVL.HUS1_LB02_GT31_MV	REAL	-50	100	-50	100	°C	0.0	Mätvärde temperatur uteluft			*)	
		HUS1_LB02_GT81_MV	AT%MB5276	:REAL;	(*	HUS1_LB02_GT81_MV	AS01	GVL.HUS1_LB02_GT81_MV	REAL	-50	100	-50	100	°C	0.0	Mätvärde temperatur frysvakt			*)	
		HUS1_LB02_VVX01_VVX	AT%MB5280	:REAL;	(*	HUS1_LB02_VVX01_VVX	AS01	GVL.HUS1_LB02_VVX01_VVX	REAL	0	100	0	100	%	0.0	Verkningsgrad VVX			*)	
		HUS1_LB02_SV21_R	AT%MB5284	:REAL;	(*	HUS1_LB02_SV21_R	AS01	GVL.HUS1_LB02_SV21_R	REAL	0	100	0	100	%	0.0	Styrsignal ventilställdon värme			*)	
		HUS2_LB03_GF41_MV	AT%MB5288	:REAL;	(*	HUS2_LB03_GF41_MV	AS01	GVL.HUS2_LB03_GF41_MV	REAL	0	4000	0	4000	l/s	0.0	Mätvärde flöde tilluft			*)	
		HUS2_LB03_GF42_MV	AT%MB5292	:REAL;	(*	HUS2_LB03_GF42_MV	AS01	GVL.HUS2_LB03_GF42_MV	REAL	0	4000	0	4000	l/s	0.0	Mätvärde flöde frånluft			*)	
		HUS2_LB03_GP11_MV	AT%MB5296	:REAL;	(*	HUS2_LB03_GP11_MV	AS01	GVL.HUS2_LB03_GP11_MV	REAL	0	1000	0	1000	Pa		Mätvärde tryck tilluft			*)	
		HUS2_LB03_GP12_MV	AT%MB5300	:REAL;	(*	HUS2_LB03_GP12_MV	AS01	GVL.HUS2_LB03_GP12_MV	REAL	0	1000	0	1000	Pa		Mätvärde tryck frånluft			*)	
		HUS2_LB03_GP61_MV	AT%MB5304	:REAL;	(*	HUS2_LB03_GP61_MV	AS01	GVL.HUS2_LB03_GP61_MV	REAL	0	1000	0	1000	Pa		Mätvärde tryckfall tilluftsfilter			*)	
		HUS2_LB03_GP61_GV	AT%MB5308	:REAL;	(*	HUS2_LB03_GP61_GV	AS01	GVL.HUS2_LB03_GP61_GV	REAL	0	1000	0	1000	Pa		Sluttryckfall tilluftsfilter			*)	
		HUS2_LB03_GP62_MV	AT%MB5312	:REAL;	(*	HUS2_LB03_GP62_MV	AS01	GVL.HUS2_LB03_GP62_MV	REAL	0	1000	0	1000	Pa		Mätvärde tryckfall frånluftsfilter			*)	
		HUS2_LB03_GP62_GV	AT%MB5316	:REAL;	(*	HUS2_LB03_GP62_GV	AS01	GVL.HUS2_LB03_GP62_GV	REAL	0	1000	0	1000	Pa		Sluttryckfall frånluftsfilter			*)	
		HUS2_LB03_TF01_R	AT%MB5320	:REAL;	(*	HUS2_LB03_TF01_R	AS01	GVL.HUS2_LB03_TF01_R	REAL	0	100	0	100	%	0.0	Styrsignal tilluftsfläkt			*)	
		HUS2_LB03_FF01_R	AT%MB5324	:REAL;	(*	HUS2_LB03_FF01_R	AS01	GVL.HUS2_LB03_FF01_R	REAL	0	100	0	100	%	0.0	Styrsignal frånluftsfläkt			*)	
		HUS2_LB03_SFP_MV	AT%MB5328	:REAL;	(*	HUS2_LB03_SFP_MV	AS01	GVL.HUS2_LB03_SFP_MV	REAL	0	100	0	100	kW/m3/s	0.0	SFP-värde			*)	
		HUS2_LB03_GT11_MV	AT%MB5332	:REAL;	(*	HUS2_LB03_GT11_MV	AS01	GVL.HUS2_LB03_GT11_MV	REAL	-50	100	-50	100	°C	0.0	Mätvärde temperatur tilluft			*)	
		HUS2_LB03_GT41_MV	AT%MB5336	:REAL;	(*	HUS2_LB03_GT41_MV	AS01	GVL.HUS2_LB03_GT41_MV	REAL	-50	100	-50	100	°C	0.0	Mätvärde temperatur frånluft			*)	
		HUS2_LB03_GT31_MV	AT%MB5340	:REAL;	(*	HUS2_LB03_GT31_MV	AS01	GVL.HUS2_LB03_GT31_MV	REAL	-50	100	-50	100	°C	0.0	Mätvärde temperatur uteluft			*)	
		HUS2_LB03_GT81_MV	AT%MB5344	:REAL;	(*	HUS2_LB03_GT81_MV	AS01	GVL.HUS2_LB03_GT81_MV	REAL	-50	100	-50	100	°C	0.0	Mätvärde temperatur frysvakt			*)	
		HUS2_LB03_VVX01_VVX	AT%MB5348	:REAL;	(*	HUS2_LB03_VVX01_VVX	AS01	GVL.HUS2_LB03_VVX01_VVX	REAL	0	100	0	100	%	0.0	Verkningsgrad VVX			*)	
		HUS2_LB03_SV21_R	AT%MB5352	:REAL;	(*	HUS2_LB03_SV21_R	AS01	GVL.HUS2_LB03_SV21_R	REAL	0	100	0	100	%	0.0	Styrsignal ventilställdon värme			*)	
		HUS3_LB04_GF41_MV	AT%MB5356	:REAL;	(*	HUS3_LB04_GF41_MV	AS01	GVL.HUS3_LB04_GF41_MV	REAL	0	4000	0	4000	l/s	0.0	Mätvärde flöde tilluft			*)	
		HUS3_LB04_GF42_MV	AT%MB5360	:REAL;	(*	HUS3_LB04_GF42_MV	AS01	GVL.HUS3_LB04_GF42_MV	REAL	0	4000	0	4000	l/s	0.0	Mätvärde flöde frånluft			*)	
		HUS3_LB04_GP11_MV	AT%MB5364	:REAL;	(*	HUS3_LB04_GP11_MV	AS01	GVL.HUS3_LB04_GP11_MV	REAL	0	1000	0	1000	Pa		Mätvärde tryck tilluft			*)	
		HUS3_LB04_GP12_MV	AT%MB5368	:REAL;	(*	HUS3_LB04_GP12_MV	AS01	GVL.HUS3_LB04_GP12_MV	REAL	0	1000	0	1000	Pa		Mätvärde tryck frånluft			*)	
		HUS3_LB04_GP61_MV	AT%MB5372	:REAL;	(*	HUS3_LB04_GP61_MV	AS01	GVL.HUS3_LB04_GP61_MV	REAL	0	1000	0	1000	Pa		Mätvärde tryckfall tilluftsfilter			*)	
		HUS3_LB04_GP61_GV	AT%MB5376	:REAL;	(*	HUS3_LB04_GP61_GV	AS01	GVL.HUS3_LB04_GP61_GV	REAL	0	1000	0	1000	Pa		Sluttryckfall tilluftsfilter			*)	
		HUS3_LB04_GP62_MV	AT%MB5380	:REAL;	(*	HUS3_LB04_GP62_MV	AS01	GVL.HUS3_LB04_GP62_MV	REAL	0	1000	0	1000	Pa		Mätvärde tryckfall frånluftsfilter			*)	
		HUS3_LB04_GP62_GV	AT%MB5384	:REAL;	(*	HUS3_LB04_GP62_GV	AS01	GVL.HUS3_LB04_GP62_GV	REAL	0	1000	0	1000	Pa		Sluttryckfall frånluftsfilter			*)	
		HUS3_LB04_TF01_R	AT%MB5388	:REAL;	(*	HUS3_LB04_TF01_R	AS01	GVL.HUS3_LB04_TF01_R	REAL	0	100	0	100	%	0.0	Styrsignal tilluftsfläkt			*)	
		HUS3_LB04_FF01_R	AT%MB5392	:REAL;	(*	HUS3_LB04_FF01_R	AS01	GVL.HUS3_LB04_FF01_R	REAL	0	100	0	100	%	0.0	Styrsignal frånluftsfläkt			*)	
		HUS3_LB04_SFP_MV	AT%MB5396	:REAL;	(*	HUS3_LB04_SFP_MV	AS01	GVL.HUS3_LB04_SFP_MV	REAL	0	100	0	100	kW/m3/s	0.0	SFP-värde			*)	
		HUS3_LB04_GT11_MV	AT%MB5400	:REAL;	(*	HUS3_LB04_GT11_MV	AS01	GVL.HUS3_LB04_GT11_MV	REAL	-50	100	-50	100	°C	0.0	Mätvärde temperatur tilluft			*)	
		HUS3_LB04_GT41_MV	AT%MB5404	:REAL;	(*	HUS3_LB04_GT41_MV	AS01	GVL.HUS3_LB04_GT41_MV	REAL	-50	100	-50	100	°C	0.0	Mätvärde temperatur frånluft			*)	
		HUS3_LB04_GT31_MV	AT%MB5408	:REAL;	(*	HUS3_LB04_GT31_MV	AS01	GVL.HUS3_LB04_GT31_MV	REAL	-50	100	-50	100	°C	0.0	Mätvärde temperatur uteluft			*)	
		HUS3_LB04_GT81_MV	AT%MB5412	:REAL;	(*	HUS3_LB04_GT81_MV	AS01	GVL.HUS3_LB04_GT81_MV	REAL	-50	100	-50	100	°C	0.0	Mätvärde temperatur frysvakt			*)	
		HUS3_LB04_VVX01_VVX	AT%MB5416	:REAL;	(*	HUS3_LB04_VVX01_VVX	AS01	GVL.HUS3_LB04_VVX01_VVX	REAL	0	100	0	100	%	0.0	Verkningsgrad VVX			*)	
		HUS3_LB04_SV21_R	AT%MB5420	:REAL;	(*	HUS3_LB04_SV21_R	AS01	GVL.HUS3_LB04_SV21_R	REAL	0	100	0	100	%	0.0	Styrsignal ventilställdon värme			*)	
		HUS3_LB05_GF41_MV	AT%MB5424	:REAL;	(*	HUS3_LB05_GF41_MV	AS01	GVL.HUS3_LB05_GF41_MV	REAL	0	4000	0	4000	l/s	0.0	Mätvärde flöde tilluft			*)	
		HUS3_LB05_GF42_MV	AT%MB5428	:REAL;	(*	HUS3_LB05_GF42_MV	AS01	GVL.HUS3_LB05_GF42_MV	REAL	0	4000	0	4000	l/s	0.0	Mätvärde flöde frånluft			*)	
		HUS3_LB05_GP11_MV	AT%MB5432	:REAL;	(*	HUS3_LB05_GP11_MV	AS01	GVL.HUS3_LB05_GP11_MV	REAL	0	1000	0	1000	Pa		Mätvärde tryck tilluft			*)	
		HUS3_LB05_GP12_MV	AT%MB5436	:REAL;	(*	HUS3_LB05_GP12_MV	AS01	GVL.HUS3_LB05_GP12_MV	REAL	0	1000	0	1000	Pa		Mätvärde tryck frånluft			*)	
		HUS3_LB05_GP61_MV	AT%MB5440	:REAL;	(*	HUS3_LB05_GP61_MV	AS01	GVL.HUS3_LB05_GP61_MV	REAL	0	1000	0	1000	Pa		Mätvärde tryckfall tilluftsfilter			*)	
		HUS3_LB05_GP61_GV	AT%MB5444	:REAL;	(*	HUS3_LB05_GP61_GV	AS01	GVL.HUS3_LB05_GP61_GV	REAL	0	1000	0	1000	Pa		Sluttryckfall tilluftsfilter			*)	
		HUS3_LB05_GP62_MV	AT%MB5448	:REAL;	(*	HUS3_LB05_GP62_MV	AS01	GVL.HUS3_LB05_GP62_MV	REAL	0	1000	0	1000	Pa		Mätvärde tryckfall frånluftsfilter			*)	
		HUS3_LB05_GP62_GV	AT%MB5452	:REAL;	(*	HUS3_LB05_GP62_GV	AS01	GVL.HUS3_LB05_GP62_GV	REAL	0	1000	0	1000	Pa		Sluttryckfall frånluftsfilter			*)	
		HUS3_LB05_TF01_R	AT%MB5456	:REAL;	(*	HUS3_LB05_TF01_R	AS01	GVL.HUS3_LB05_TF01_R	REAL	0	100	0	100	%	0.0	Styrsignal tilluftsfläkt			*)	
		HUS3_LB05_FF01_R	AT%MB5460	:REAL;	(*	HUS3_LB05_FF01_R	AS01	GVL.HUS3_LB05_FF01_R	REAL	0	100	0	100	%	0.0	Styrsignal frånluftsfläkt			*)	
		HUS3_LB05_SFP_MV	AT%MB5464	:REAL;	(*	HUS3_LB05_SFP_MV	AS01	GVL.HUS3_LB05_SFP_MV	REAL	0	100	0	100	kW/m3/s	0.0	SFP-värde			*)	
		HUS3_LB05_GT11_MV	AT%MB5468	:REAL;	(*	HUS3_LB05_GT11_MV	AS01	GVL.HUS3_LB05_GT11_MV	REAL	-50	100	-50	100	°C	0.0	Mätvärde temperatur tilluft			*)	
		HUS3_LB05_GT41_MV	AT%MB5472	:REAL;	(*	HUS3_LB05_GT41_MV	AS01	GVL.HUS3_LB05_GT41_MV	REAL	-50	100	-50	100	°C	0.0	Mätvärde temperatur frånluft			*)	
		HUS3_LB05_GT31_MV	AT%MB5476	:REAL;	(*	HUS3_LB05_GT31_MV	AS01	GVL.HUS3_LB05_GT31_MV	REAL	-50	100	-50	100	°C	0.0	Mätvärde temperatur uteluft			*)	
		HUS3_LB05_GT81_MV	AT%MB5480	:REAL;	(*	HUS3_LB05_GT81_MV	AS01	GVL.HUS3_LB05_GT81_MV	REAL	-50	100	-50	100	°C	0.0	Mätvärde temperatur frysvakt			*)	
		HUS3_LB05_VVX01_VVX	AT%MB5484	:REAL;	(*	HUS3_LB05_VVX01_VVX	AS01	GVL.HUS3_LB05_VVX01_VVX	REAL	0	100	0	100	%	0.0	Verkningsgrad VVX			*)	
		HUS3_LB05_SV21_R	AT%MB5488	:REAL;	(*	HUS3_LB05_SV21_R	AS01	GVL.HUS3_LB05_SV21_R	REAL	0	100	0	100	%	0.0	Styrsignal ventilställdon värme			*)	
		HUS1_LB06_GF41_MV	AT%MB5492	:REAL;	(*	HUS1_LB06_GF41_MV	AS01	GVL.HUS1_LB06_GF41_MV	REAL	0	4000	0	4000	l/s	0.0	Mätvärde flöde tilluft			*)	
		HUS1_LB06_GF42_MV	AT%MB5496	:REAL;	(*	HUS1_LB06_GF42_MV	AS01	GVL.HUS1_LB06_GF42_MV	REAL	0	4000	0	4000	l/s	0.0	Mätvärde flöde frånluft			*)	
		HUS1_LB06_GP11_MV	AT%MB5500	:REAL;	(*	HUS1_LB06_GP11_MV	AS01	GVL.HUS1_LB06_GP11_MV	REAL	0	1000	0	1000	Pa		Mätvärde tryck tilluft			*)	
		HUS1_LB06_GP12_MV	AT%MB5504	:REAL;	(*	HUS1_LB06_GP12_MV	AS01	GVL.HUS1_LB06_GP12_MV	REAL	0	1000	0	1000	Pa		Mätvärde tryck frånluft			*)	
		HUS1_LB06_GP61_MV	AT%MB5508	:REAL;	(*	HUS1_LB06_GP61_MV	AS01	GVL.HUS1_LB06_GP61_MV	REAL	0	1000	0	1000	Pa		Mätvärde tryckfall tilluftsfilter			*)	
		HUS1_LB06_GP61_GV	AT%MB5512	:REAL;	(*	HUS1_LB06_GP61_GV	AS01	GVL.HUS1_LB06_GP61_GV	REAL	0	1000	0	1000	Pa		Sluttryckfall tilluftsfilter			*)	
		HUS1_LB06_GP62_MV	AT%MB5516	:REAL;	(*	HUS1_LB06_GP62_MV	AS01	GVL.HUS1_LB06_GP62_MV	REAL	0	1000	0	1000	Pa		Mätvärde tryckfall frånluftsfilter			*)	
		HUS1_LB06_GP62_GV	AT%MB5520	:REAL;	(*	HUS1_LB06_GP62_GV	AS01	GVL.HUS1_LB06_GP62_GV	REAL	0	1000	0	1000	Pa		Sluttryckfall frånluftsfilter			*)	
		HUS1_LB06_TF01_R	AT%MB5524	:REAL;	(*	HUS1_LB06_TF01_R	AS01	GVL.HUS1_LB06_TF01_R	REAL	0	100	0	100	%	0.0	Styrsignal tilluftsfläkt			*)	
		HUS1_LB06_FF01_R	AT%MB5528	:REAL;	(*	HUS1_LB06_FF01_R	AS01	GVL.HUS1_LB06_FF01_R	REAL	0	100	0	100	%	0.0	Styrsignal frånluftsfläkt			*)	
		HUS1_LB06_SFP_MV	AT%MB5532	:REAL;	(*	HUS1_LB06_SFP_MV	AS01	GVL.HUS1_LB06_SFP_MV	REAL	0	100	0	100	kW/m3/s	0.0	SFP-värde			*)	
		HUS1_LB06_GT11_MV	AT%MB5536	:REAL;	(*	HUS1_LB06_GT11_MV	AS01	GVL.HUS1_LB06_GT11_MV	REAL	-50	100	-50	100	°C	0.0	Mätvärde temperatur tilluft			*)	
		HUS1_LB06_GT41_MV	AT%MB5540	:REAL;	(*	HUS1_LB06_GT41_MV	AS01	GVL.HUS1_LB06_GT41_MV	REAL	-50	100	-50	100	°C	0.0	Mätvärde temperatur frånluft			*)	
		HUS1_LB06_GT31_MV	AT%MB5544	:REAL;	(*	HUS1_LB06_GT31_MV	AS01	GVL.HUS1_LB06_GT31_MV	REAL	-50	100	-50	100	°C	0.0	Mätvärde temperatur uteluft			*)	
		HUS1_LB06_GT81_MV	AT%MB5548	:REAL;	(*	HUS1_LB06_GT81_MV	AS01	GVL.HUS1_LB06_GT81_MV	REAL	-50	100	-50	100	°C	0.0	Mätvärde temperatur frysvakt			*)	
		HUS1_LB06_VVX01_VVX	AT%MB5552	:REAL;	(*	HUS1_LB06_VVX01_VVX	AS01	GVL.HUS1_LB06_VVX01_VVX	REAL	0	100	0	100	%	0.0	Verkningsgrad VVX			*)	
		HUS1_LB06_SV21_R	AT%MB5556	:REAL;	(*	HUS1_LB06_SV21_R	AS01	GVL.HUS1_LB06_SV21_R	REAL	0	100	0	100	%	0.0	Styrsignal ventilställdon värme			*)	


END_VAR

(* Global variable list: xOvrigt/SystemTime *)
VAR_GLOBAL
(****************************************************************************************************)
(****************************************************************************************************)
(*SystemTime*)
	stSystemTime				: 	TIMESTRUCT;
	dtSystemTime				: 	DT;
	uiYear						: 	UINT;
	uiMonth						: 	UINT;
	uiDay						: 	UINT;
	uiDayOfWeek				: 	UINT;
	uiHour						: 	UINT;
	uiMinute						: 	UINT;
	uiSecond					: 	UINT;
	uiMilliseconds				: 	UINT;
(****************************************************************************************************)
(*SystemTaskInfo*)
	tTaskCycleTime			: 	TIME;			(* task cycle time *)
	tLastExecCycleTime		:	TIME;			(* latest cycle time *)
(****************************************************************************************************)
END_VAR

